LIN {X 0,Y 573.961,Z 401.905,A -85,B 0,C 180,E1 -2264.781,E2 -2264.781} C_VEL
LIN {X 0,Y 574.137,Z 387.873,A -85,B 0,C 180,E1 -2265.623,E2 -2265.623} C_VEL
LIN {X 0,Y 574.369,Z 373.799,A -85,B 0,C 180,E1 -2266.3,E2 -2266.3} C_VEL
LIN {X 0,Y 574.566,Z 359.304,A -85,B 0,C 180,E1 -2266.843,E2 -2266.843} C_VEL
LIN {X 0,Y 574.72,Z 343.895,A -85,B 0,C 180,E1 -2267.263,E2 -2267.263} C_VEL
LIN {X 0,Y 574.806,Z 328.514,A -85,B 0,C 180,E1 -2267.533,E2 -2267.533} C_VEL
LIN {X 0,Y 575.107,Z 176.129,A -85,B 0,C 180,E1 -2269.49,E2 -2269.49} C_VEL
LIN {X 0,Y 573.982,Z 170.376,A -85,B 0,C 180,E1 -2269.621,E2 -2269.621} C_VEL
LIN {X 0,Y 574.205,Z 150.282,A -85,B 0,C 180,E1 -2272.109,E2 -2272.109} C_VEL
LIN {X 0,Y 574.45,Z 130.828,A -85,B 0,C 180,E1 -2274.58,E2 -2274.58} C_VEL
LIN {X 0,Y 573.276,Z 124.83,A -85,B 0,C 180,E1 -2275.433,E2 -2275.433} C_VEL
LIN {X 0,Y 573.251,Z 124.698,A -85,B 0,C 180,E1 -2278.029,E2 -2278.029} C_VEL
LIN {X 0,Y 573.247,Z 124.707,A -85,B 0,C 180,E1 -2280.176,E2 -2280.176} C_VEL
LIN {X 0,Y 573.254,Z 124.699,A -85,B 0,C 180,E1 -2282.645,E2 -2282.645} C_VEL
LIN {X 0,Y 573.206,Z 124.704,A -85,B 0,C 180,E1 -2285.188,E2 -2285.188} C_VEL
LIN {X 0,Y 573.237,Z 124.707,A -85,B 0,C 180,E1 -2287.808,E2 -2287.808} C_VEL
LIN {X 0,Y 573.245,Z 124.7,A -85,B 0,C 180,E1 -2290.525,E2 -2290.525} C_VEL
LIN {X 0,Y 573.237,Z 124.702,A -85,B 0,C 180,E1 -2293.359,E2 -2293.359} C_VEL
LIN {X 0,Y 573.246,Z 124.701,A -85,B 0,C 180,E1 -2296.331,E2 -2296.331} C_VEL
LIN {X 0,Y 573.23,Z 124.698,A -85,B 0,C 180,E1 -2298.543,E2 -2298.543} C_VEL
LIN {X 0,Y 573.242,Z 124.702,A -85,B 0,C 180,E1 -2301.299,E2 -2301.299} C_VEL
LIN {X 0,Y 573.213,Z 124.704,A -85,B 0,C 180,E1 -2304.019,E2 -2304.019} C_VEL
LIN {X 0,Y 573.234,Z 124.694,A -85,B 0,C 180,E1 -2306.516,E2 -2306.516} C_VEL
LIN {X 0,Y 573.225,Z 124.703,A -85,B 0,C 180,E1 -2309.119,E2 -2309.119} C_VEL
LIN {X 0,Y 573.236,Z 124.707,A -85,B 0,C 180,E1 -2311.436,E2 -2311.436} C_VEL
LIN {X 0,Y 573.26,Z 124.697,A -85,B 0,C 180,E1 -2313.81,E2 -2313.81} C_VEL
LIN {X 0,Y 573.223,Z 124.702,A -85,B 0,C 180,E1 -2316.134,E2 -2316.134} C_VEL
LIN {X 0,Y 573.249,Z 124.706,A -85,B 0,C 180,E1 -2319.174,E2 -2319.174} C_VEL
LIN {X 0,Y 573.214,Z 124.707,A -85,B 0,C 180,E1 -2321.411,E2 -2321.411} C_VEL
LIN {X 0,Y 573.24,Z 124.699,A -85,B 0,C 180,E1 -2323.621,E2 -2323.621} C_VEL
LIN {X 0,Y 573.224,Z 124.705,A -85,B 0,C 180,E1 -2326.529,E2 -2326.529} C_VEL
LIN {X 0,Y 573.265,Z 124.705,A -85,B 0,C 180,E1 -2328.745,E2 -2328.745} C_VEL
LIN {X 0,Y 573.253,Z 124.697,A -85,B 0,C 180,E1 -2331.54,E2 -2331.54} C_VEL
LIN {X 0,Y 573.297,Z 124.697,A -85,B 0,C 180,E1 -2334.372,E2 -2334.372} C_VEL
LIN {X 0,Y 573.312,Z 124.69,A -85,B 0,C 180,E1 -2337.893,E2 -2337.893} C_VEL
LIN {X 0,Y 573.329,Z 124.693,A -85,B 0,C 180,E1 -2340.702,E2 -2340.702} C_VEL
LIN {X 0,Y 573.293,Z 124.695,A -85,B 0,C 180,E1 -2342.811,E2 -2342.811} C_VEL
LIN {X 0,Y 573.283,Z 124.695,A -85,B 0,C 180,E1 -2345.628,E2 -2345.628} C_VEL
LIN {X 0,Y 573.28,Z 124.699,A -85,B 0,C 180,E1 -2348.46,E2 -2348.46} C_VEL
LIN {X 0,Y 573.275,Z 124.695,A -85,B 0,C 180,E1 -2351.312,E2 -2351.312} C_VEL
LIN {X 0,Y 573.273,Z 124.698,A -85,B 0,C 180,E1 -2354.42,E2 -2354.42} C_VEL
LIN {X 0,Y 573.196,Z 124.705,A -85,B 0,C 180,E1 -2357.114,E2 -2357.114} C_VEL
LIN {X 0,Y 573.267,Z 124.696,A -85,B 0,C 180,E1 -2359.33,E2 -2359.33} C_VEL
LIN {X 0,Y 573.221,Z 124.705,A -85,B 0,C 180,E1 -2362.339,E2 -2362.339} C_VEL
LIN {X 0,Y 573.208,Z 124.704,A -85,B 0,C 180,E1 -2364.372,E2 -2364.372} C_VEL
LIN {X 0,Y 572.57,Z 124.783,A -85,B 0,C 180,E1 -2364.959,E2 -2364.959} C_VEL
LIN {X 0,Y 569.729,Z 125.144,A -85,B 0,C 180,E1 -2365.91,E2 -2365.91} C_VEL
LIN {X 0,Y 567.305,Z 125.446,A -85,B 0,C 180,E1 -2366.676,E2 -2366.676} C_VEL
LIN {X 0,Y 566.254,Z 125.574,A -85,B 0,C 180,E1 -2367.267,E2 -2367.267} C_VEL
LIN {X 0,Y 566.163,Z 125.584,A -85,B 0,C 180,E1 -2367.467,E2 -2367.467} C_VEL
LIN {X 0,Y 566.17,Z 125.584,A -85,B 0,C 180,E1 -2369.771,E2 -2369.771} C_VEL
LIN {X 0,Y 566.193,Z 125.57,A -85,B 0,C 180,E1 -2372.428,E2 -2372.428} C_VEL
LIN {X 0,Y 566.167,Z 125.581,A -85,B 0,C 180,E1 -2374.987,E2 -2374.987} C_VEL
LIN {X 0,Y 566.191,Z 125.585,A -85,B 0,C 180,E1 -2377.461,E2 -2377.461} C_VEL
LIN {X 0,Y 566.206,Z 125.57,A -85,B 0,C 180,E1 -2380.199,E2 -2380.199} C_VEL
LIN {X 0,Y 566.179,Z 125.584,A -85,B 0,C 180,E1 -2383.056,E2 -2383.056} C_VEL
LIN {X 0,Y 566.156,Z 125.579,A -85,B 0,C 180,E1 -2386.053,E2 -2386.053} C_VEL
LIN {X 0,Y 566.164,Z 125.587,A -85,B 0,C 180,E1 -2388.859,E2 -2388.859} C_VEL
LIN {X 0,Y 566.202,Z 125.581,A -85,B 0,C 180,E1 -2391.443,E2 -2391.443} C_VEL
LIN {X 0,Y 566.136,Z 125.585,A -85,B 0,C 180,E1 -2394.306,E2 -2394.306} C_VEL
LIN {X 0,Y 566.193,Z 125.585,A -85,B 0,C 180,E1 -2396.896,E2 -2396.896} C_VEL
LIN {X 0,Y 566.15,Z 125.578,A -85,B 0,C 180,E1 -2399.405,E2 -2399.405} C_VEL
LIN {X 0,Y 566.141,Z 125.586,A -85,B 0,C 180,E1 -2401.854,E2 -2401.854} C_VEL
LIN {X 0,Y 566.175,Z 125.585,A -85,B 0,C 180,E1 -2404.249,E2 -2404.249} C_VEL
LIN {X 0,Y 566.208,Z 125.751,A -85,B 0,C 180,E1 -2405.405,E2 -2405.405} C_VEL
LIN {X 0,Y 567.351,Z 131.059,A -85,B 0,C 180,E1 -2406.212,E2 -2406.212} C_VEL
LIN {X 0,Y 567.208,Z 146.629,A -85,B 0,C 180,E1 -2408.324,E2 -2408.324} C_VEL
LIN {X 0,Y 567.018,Z 160.677,A -85,B 0,C 180,E1 -2410.172,E2 -2410.172} C_VEL
LIN {X 0,Y 568.504,Z 168.273,A -85,B 0,C 180,E1 -2410.348,E2 -2410.348} C_VEL
LIN {X 0,Y 567.975,Z 326.141,A -85,B 0,C 180,E1 -2412.412,E2 -2412.412} C_VEL
LIN {X 0,Y 567.824,Z 341.766,A -85,B 0,C 180,E1 -2412.766,E2 -2412.766} C_VEL
LIN {X 0,Y 567.638,Z 357.075,A -85,B 0,C 180,E1 -2413.27,E2 -2413.27} C_VEL
LIN {X 0,Y 567.408,Z 371.73,A -85,B 0,C 180,E1 -2413.91,E2 -2413.91} C_VEL
LIN {X 0,Y 567.132,Z 385.048,A -85,B 0,C 180,E1 -2414.64,E2 -2414.64} C_VEL
LIN {X 0,Y 566.918,Z 397.981,A -85,B 0,C 180,E1 -2415.508,E2 -2415.508} C_VEL
LIN {X 0,Y 566.653,Z 410.889,A -85,B 0,C 180,E1 -2416.553,E2 -2416.553} C_VEL
LIN {X 0,Y 566.462,Z 422.085,A -85,B 0,C 180,E1 -2417.642,E2 -2417.642} C_VEL
LIN {X 0,Y 566.264,Z 432.178,A -85,B 0,C 180,E1 -2418.81,E2 -2418.81} C_VEL
LIN {X 0,Y 566.132,Z 442.003,A -85,B 0,C 180,E1 -2420.172,E2 -2420.172} C_VEL
LIN {X 0,Y 566.063,Z 449.494,A -85,B 0,C 180,E1 -2421.432,E2 -2421.432} C_VEL
LIN {X 0,Y 565.975,Z 456.499,A -85,B 0,C 180,E1 -2422.867,E2 -2422.867} C_VEL
LIN {X 0,Y 565.982,Z 462.009,A -85,B 0,C 180,E1 -2424.299,E2 -2424.299} C_VEL
LIN {X 0,Y 565.913,Z 466.177,A -85,B 0,C 180,E1 -2425.727,E2 -2425.727} C_VEL
LIN {X 0,Y 565.872,Z 469.112,A -85,B 0,C 180,E1 -2427.152,E2 -2427.152} C_VEL
LIN {X 0,Y 565.842,Z 470.879,A -85,B 0,C 180,E1 -2428.577,E2 -2428.577} C_VEL
LIN {X 0,Y 565.837,Z 471.496,A -85,B 0,C 180,E1 -2430,E2 -2430} C_VEL
LIN {X 0,Y 565.843,Z 470.941,A -85,B 0,C 180,E1 -2431.423,E2 -2431.423} C_VEL
LIN {X 0,Y 565.874,Z 469.257,A -85,B 0,C 180,E1 -2432.848,E2 -2432.848} C_VEL
LIN {X 0,Y 565.913,Z 466.404,A -85,B 0,C 180,E1 -2434.273,E2 -2434.273} C_VEL
LIN {X 0,Y 565.975,Z 462.318,A -85,B 0,C 180,E1 -2435.701,E2 -2435.701} C_VEL
LIN {X 0,Y 565.975,Z 456.903,A -85,B 0,C 180,E1 -2437.133,E2 -2437.133} C_VEL
LIN {X 0,Y 566.061,Z 450.002,A -85,B 0,C 180,E1 -2438.568,E2 -2438.568} C_VEL
LIN {X 0,Y 566.177,Z 441.393,A -85,B 0,C 180,E1 -2440.008,E2 -2440.008} C_VEL
LIN {X 0,Y 566.25,Z 432.953,A -85,B 0,C 180,E1 -2441.183,E2 -2441.183} C_VEL
LIN {X 0,Y 566.43,Z 422.913,A -85,B 0,C 180,E1 -2442.359,E2 -2442.359} C_VEL
LIN {X 0,Y 566.669,Z 410.869,A -85,B 0,C 180,E1 -2443.538,E2 -2443.538} C_VEL
LIN {X 0,Y 566.879,Z 399.242,A -85,B 0,C 180,E1 -2444.488,E2 -2444.488} C_VEL
LIN {X 0,Y 567.09,Z 386.467,A -85,B 0,C 180,E1 -2445.361,E2 -2445.361} C_VEL
LIN {X 0,Y 567.361,Z 373.456,A -85,B 0,C 180,E1 -2446.091,E2 -2446.091} C_VEL
LIN {X 0,Y 567.571,Z 359.261,A -85,B 0,C 180,E1 -2446.732,E2 -2446.732} C_VEL
LIN {X 0,Y 567.791,Z 344.711,A -85,B 0,C 180,E1 -2447.235,E2 -2447.235} C_VEL
LIN {X 0,Y 567.93,Z 329.3,A -85,B 0,C 180,E1 -2447.615,E2 -2447.615} C_VEL
LIN {X 0,Y 568.045,Z 307.857,A -85,B 0,C 180,E1 -2447.933,E2 -2447.933} C_VEL
LIN {X 0,Y 568.445,Z 167.858,A -85,B 0,C 180,E1 -2449.75,E2 -2449.75} C_VEL
LIN {X 0,Y 567.012,Z 160.622,A -85,B 0,C 180,E1 -2449.921,E2 -2449.921} C_VEL
LIN {X 0,Y 567.371,Z 139.147,A -85,B 0,C 180,E1 -2452.774,E2 -2452.774} C_VEL
LIN {X 0,Y 567.419,Z 131.697,A -85,B 0,C 180,E1 -2453.788,E2 -2453.788} C_VEL
LIN {X 0,Y 566.213,Z 125.822,A -85,B 0,C 180,E1 -2454.668,E2 -2454.668} C_VEL
LIN {X 0,Y 566.164,Z 125.581,A -85,B 0,C 180,E1 -2456.65,E2 -2456.65} C_VEL
LIN {X 0,Y 566.144,Z 125.58,A -85,B 0,C 180,E1 -2459.772,E2 -2459.772} C_VEL
LIN {X 0,Y 566.177,Z 125.581,A -85,B 0,C 180,E1 -2462.425,E2 -2462.425} C_VEL
LIN {X 0,Y 566.159,Z 125.589,A -85,B 0,C 180,E1 -2464.986,E2 -2464.986} C_VEL
LIN {X 0,Y 566.189,Z 125.582,A -85,B 0,C 180,E1 -2467.462,E2 -2467.462} C_VEL
LIN {X 0,Y 566.166,Z 125.579,A -85,B 0,C 180,E1 -2470.203,E2 -2470.203} C_VEL
LIN {X 0,Y 566.177,Z 125.584,A -85,B 0,C 180,E1 -2473.057,E2 -2473.057} C_VEL
LIN {X 0,Y 566.157,Z 125.582,A -85,B 0,C 180,E1 -2476.053,E2 -2476.053} C_VEL
LIN {X 0,Y 566.151,Z 125.584,A -85,B 0,C 180,E1 -2478.858,E2 -2478.858} C_VEL
LIN {X 0,Y 566.199,Z 125.575,A -85,B 0,C 180,E1 -2481.444,E2 -2481.444} C_VEL
LIN {X 0,Y 566.141,Z 125.59,A -85,B 0,C 180,E1 -2484.306,E2 -2484.306} C_VEL
LIN {X 0,Y 566.196,Z 125.573,A -85,B 0,C 180,E1 -2486.896,E2 -2486.896} C_VEL
LIN {X 0,Y 566.168,Z 125.576,A -85,B 0,C 180,E1 -2489.406,E2 -2489.406} C_VEL
LIN {X 0,Y 566.15,Z 125.585,A -85,B 0,C 180,E1 -2491.854,E2 -2491.854} C_VEL
LIN {X 0,Y 566.193,Z 125.585,A -85,B 0,C 180,E1 -2494.25,E2 -2494.25} C_VEL
LIN {X 0,Y 566.164,Z 125.581,A -85,B 0,C 180,E1 -2497.368,E2 -2497.368} C_VEL
LIN {X 0,Y 566.194,Z 125.579,A -85,B 0,C 180,E1 -2499.662,E2 -2499.662} C_VEL
LIN {X 0,Y 566.17,Z 125.586,A -85,B 0,C 180,E1 -2501.921,E2 -2501.921} C_VEL
LIN {X 0,Y 566.188,Z 125.576,A -85,B 0,C 180,E1 -2504.89,E2 -2504.89} C_VEL
LIN {X 0,Y 566.213,Z 125.582,A -85,B 0,C 180,E1 -2507.818,E2 -2507.818} C_VEL
LIN {X 0,Y 566.172,Z 125.585,A -85,B 0,C 180,E1 -2509.992,E2 -2509.992} C_VEL
LIN {X 0,Y 566.213,Z 125.574,A -85,B 0,C 180,E1 -2512.87,E2 -2512.87} C_VEL
LIN {X 0,Y 566.267,Z 125.569,A -85,B 0,C 180,E1 -2515.016,E2 -2515.016} C_VEL
LIN {X 0,Y 566.284,Z 125.569,A -85,B 0,C 180,E1 -2517.866,E2 -2517.866} C_VEL
LIN {X 0,Y 566.289,Z 125.565,A -85,B 0,C 180,E1 -2520.711,E2 -2520.711} C_VEL
LIN {X 0,Y 566.258,Z 125.569,A -85,B 0,C 180,E1 -2522.846,E2 -2522.846} C_VEL
LIN {X 0,Y 566.262,Z 125.573,A -85,B 0,C 180,E1 -2525.698,E2 -2525.698} C_VEL
LIN {X 0,Y 566.204,Z 125.575,A -85,B 0,C 180,E1 -2528.566,E2 -2528.566} C_VEL
LIN {X 0,Y 566.245,Z 125.577,A -85,B 0,C 180,E1 -2531.454,E2 -2531.454} C_VEL
LIN {X 0,Y 566.221,Z 125.574,A -85,B 0,C 180,E1 -2534.5,E2 -2534.5} C_VEL
LIN {X 0,Y 566.19,Z 125.583,A -85,B 0,C 180,E1 -2537.332,E2 -2537.332} C_VEL
LIN {X 0,Y 566.203,Z 125.577,A -85,B 0,C 180,E1 -2539.581,E2 -2539.581} C_VEL
LIN {X 0,Y 566.189,Z 125.577,A -85,B 0,C 180,E1 -2541.863,E2 -2541.863} C_VEL
LIN {X 0,Y 566.185,Z 125.583,A -85,B 0,C 180,E1 -2545.022,E2 -2545.022} C_VEL
LIN {X 0,Y 566.209,Z 125.577,A -85,B 0,C 180,E1 -2547.339,E2 -2547.339} C_VEL
LIN {X 0,Y 566.198,Z 125.576,A -85,B 0,C 180,E1 -2549.769,E2 -2549.769} C_VEL
LIN {X 0,Y 566.204,Z 125.578,A -85,B 0,C 180,E1 -2552.429,E2 -2552.429} C_VEL
LIN {X 0,Y 566.181,Z 125.581,A -85,B 0,C 180,E1 -2554.989,E2 -2554.989} C_VEL
LIN {X 0,Y 566.197,Z 125.577,A -85,B 0,C 180,E1 -2557.461,E2 -2557.461} C_VEL
LIN {X 0,Y 566.208,Z 125.579,A -85,B 0,C 180,E1 -2560.199,E2 -2560.199} C_VEL
LIN {X 0,Y 566.203,Z 125.577,A -85,B 0,C 180,E1 -2563.054,E2 -2563.054} C_VEL
LIN {X 0,Y 566.195,Z 125.582,A -85,B 0,C 180,E1 -2566.049,E2 -2566.049} C_VEL
LIN {X 0,Y 566.205,Z 125.576,A -85,B 0,C 180,E1 -2569.214,E2 -2569.214} C_VEL
LIN {X 0,Y 566.19,Z 125.58,A -85,B 0,C 180,E1 -2571.637,E2 -2571.637} C_VEL
LIN {X 0,Y 566.163,Z 125.586,A -85,B 0,C 180,E1 -2574.308,E2 -2574.308} C_VEL
LIN {X 0,Y 566.221,Z 125.572,A -85,B 0,C 180,E1 -2576.898,E2 -2576.898} C_VEL
LIN {X 0,Y 566.181,Z 125.58,A -85,B 0,C 180,E1 -2579.407,E2 -2579.407} C_VEL
LIN {X 0,Y 566.213,Z 125.574,A -85,B 0,C 180,E1 -2581.857,E2 -2581.857} C_VEL
LIN {X 0,Y 566.233,Z 125.711,A -85,B 0,C 180,E1 -2584.357,E2 -2584.357} C_VEL
LIN {X 0,Y 567.584,Z 132.266,A -85,B 0,C 180,E1 -2585.298,E2 -2585.298} C_VEL
LIN {X 0,Y 567.325,Z 151.718,A -85,B 0,C 180,E1 -2587.8,E2 -2587.8} C_VEL
LIN {X 0,Y 567.06,Z 170.307,A -85,B 0,C 180,E1 -2590.126,E2 -2590.126} C_VEL
LIN {X 0,Y 568.525,Z 178.114,A -85,B 0,C 180,E1 -2590.301,E2 -2590.301} C_VEL
LIN {X 0,Y 567.999,Z 335.64,A -85,B 0,C 180,E1 -2592.359,E2 -2592.359} C_VEL
LIN {X 0,Y 567.86,Z 351.148,A -85,B 0,C 180,E1 -2592.705,E2 -2592.705} C_VEL
LIN {X 0,Y 567.634,Z 365.796,A -85,B 0,C 180,E1 -2593.177,E2 -2593.177} C_VEL
LIN {X 0,Y 567.403,Z 380.776,A -85,B 0,C 180,E1 -2593.818,E2 -2593.818} C_VEL
LIN {X 0,Y 567.147,Z 394.249,A -85,B 0,C 180,E1 -2594.548,E2 -2594.548} C_VEL
LIN {X 0,Y 566.932,Z 406.519,A -85,B 0,C 180,E1 -2595.359,E2 -2595.359} C_VEL
LIN {X 0,Y 566.672,Z 419.292,A -85,B 0,C 180,E1 -2596.37,E2 -2596.37} C_VEL
LIN {X 0,Y 566.491,Z 430.749,A -85,B 0,C 180,E1 -2597.461,E2 -2597.461} C_VEL
LIN {X 0,Y 566.268,Z 441.311,A -85,B 0,C 180,E1 -2598.659,E2 -2598.659} C_VEL
LIN {X 0,Y 566.208,Z 449.855,A -85,B 0,C 180,E1 -2599.812,E2 -2599.812} C_VEL
LIN {X 0,Y 566.057,Z 457.735,A -85,B 0,C 180,E1 -2601.072,E2 -2601.072} C_VEL
LIN {X 0,Y 565.997,Z 465.09,A -85,B 0,C 180,E1 -2602.508,E2 -2602.508} C_VEL
LIN {X 0,Y 565.959,Z 470.922,A -85,B 0,C 180,E1 -2603.941,E2 -2603.941} C_VEL
LIN {X 0,Y 565.867,Z 474.386,A -85,B 0,C 180,E1 -2605.012,E2 -2605.012} C_VEL
LIN {X 0,Y 565.91,Z 477.889,A -85,B 0,C 180,E1 -2606.44,E2 -2606.44} C_VEL
LIN {X 0,Y 565.839,Z 480.191,A -85,B 0,C 180,E1 -2607.865,E2 -2607.865} C_VEL
LIN {X 0,Y 565.836,Z 481.349,A -85,B 0,C 180,E1 -2609.288,E2 -2609.288} C_VEL
LIN {X 0,Y 565.836,Z 481.348,A -85,B 0,C 180,E1 -2610.712,E2 -2610.712} C_VEL
LIN {X 0,Y 565.839,Z 480.189,A -85,B 0,C 180,E1 -2612.135,E2 -2612.135} C_VEL
LIN {X 0,Y 565.91,Z 477.886,A -85,B 0,C 180,E1 -2613.56,E2 -2613.56} C_VEL
LIN {X 0,Y 565.867,Z 474.386,A -85,B 0,C 180,E1 -2614.988,E2 -2614.988} C_VEL
LIN {X 0,Y 565.942,Z 469.609,A -85,B 0,C 180,E1 -2616.417,E2 -2616.417} C_VEL
LIN {X 0,Y 566.014,Z 463.422,A -85,B 0,C 180,E1 -2617.85,E2 -2617.85} C_VEL
LIN {X 0,Y 566.071,Z 455.646,A -85,B 0,C 180,E1 -2619.288,E2 -2619.288} C_VEL
LIN {X 0,Y 566.239,Z 447.368,A -85,B 0,C 180,E1 -2620.549,E2 -2620.549} C_VEL
LIN {X 0,Y 566.367,Z 437.391,A -85,B 0,C 180,E1 -2621.815,E2 -2621.815} C_VEL
LIN {X 0,Y 566.586,Z 427.186,A -85,B 0,C 180,E1 -2622.901,E2 -2622.901} C_VEL
LIN {X 0,Y 566.799,Z 415.019,A -85,B 0,C 180,E1 -2623.992,E2 -2623.992} C_VEL
LIN {X 0,Y 567.039,Z 402.337,A -85,B 0,C 180,E1 -2624.936,E2 -2624.936} C_VEL
LIN {X 0,Y 567.227,Z 389.508,A -85,B 0,C 180,E1 -2625.726,E2 -2625.726} C_VEL
LIN {X 0,Y 567.494,Z 374.824,A -85,B 0,C 180,E1 -2626.457,E2 -2626.457} C_VEL
LIN {X 0,Y 567.755,Z 360.613,A -85,B 0,C 180,E1 -2627.004,E2 -2627.004} C_VEL
LIN {X 0,Y 567.874,Z 346.147,A -85,B 0,C 180,E1 -2627.421,E2 -2627.421} C_VEL
LIN {X 0,Y 568.02,Z 330.546,A -85,B 0,C 180,E1 -2627.719,E2 -2627.719} C_VEL
LIN {X 0,Y 568.449,Z 177.138,A -85,B 0,C 180,E1 -2629.714,E2 -2629.714} C_VEL
LIN {X 0,Y 567.081,Z 170.463,A -85,B 0,C 180,E1 -2629.865,E2 -2629.865} C_VEL
LIN {X 0,Y 567.148,Z 159.516,A -85,B 0,C 180,E1 -2631.211,E2 -2631.211} C_VEL
LIN {X 0,Y 567.573,Z 138.034,A -85,B 0,C 180,E1 -2633.952,E2 -2633.952} C_VEL
LIN {X 0,Y 567.614,Z 132.265,A -85,B 0,C 180,E1 -2634.701,E2 -2634.701} C_VEL
LIN {X 0,Y 566.227,Z 125.676,A -85,B 0,C 180,E1 -2635.664,E2 -2635.664} C_VEL
LIN {X 0,Y 566.203,Z 125.576,A -85,B 0,C 180,E1 -2638.202,E2 -2638.202} C_VEL
LIN {X 0,Y 566.191,Z 125.575,A -85,B 0,C 180,E1 -2641.076,E2 -2641.076} C_VEL
LIN {X 0,Y 566.212,Z 125.578,A -85,B 0,C 180,E1 -2643.734,E2 -2643.734} C_VEL
LIN {X 0,Y 566.2,Z 125.579,A -85,B 0,C 180,E1 -2646.57,E2 -2646.57} C_VEL
LIN {X 0,Y 566.223,Z 125.578,A -85,B 0,C 180,E1 -2649.687,E2 -2649.687} C_VEL
LIN {X 0,Y 566.202,Z 125.575,A -85,B 0,C 180,E1 -2652.917,E2 -2652.917} C_VEL
LIN {X 0,Y 566.199,Z 125.582,A -85,B 0,C 180,E1 -2656.049,E2 -2656.049} C_VEL
LIN {X 0,Y 566.204,Z 125.576,A -85,B 0,C 180,E1 -2659.215,E2 -2659.215} C_VEL
LIN {X 0,Y 566.187,Z 125.587,A -85,B 0,C 180,E1 -2661.637,E2 -2661.637} C_VEL
LIN {X 0,Y 566.163,Z 125.58,A -85,B 0,C 180,E1 -2664.308,E2 -2664.308} C_VEL
LIN {X 0,Y 566.202,Z 125.571,A -85,B 0,C 180,E1 -2666.897,E2 -2666.897} C_VEL
LIN {X 0,Y 566.176,Z 125.586,A -85,B 0,C 180,E1 -2669.407,E2 -2669.407} C_VEL
LIN {X 0,Y 566.196,Z 125.579,A -85,B 0,C 180,E1 -2671.857,E2 -2671.857} C_VEL
LIN {X 0,Y 566.21,Z 125.573,A -85,B 0,C 180,E1 -2674.251,E2 -2674.251} C_VEL
LIN {X 0,Y 566.169,Z 125.584,A -85,B 0,C 180,E1 -2676.72,E2 -2676.72} C_VEL
LIN {X 0,Y 566.206,Z 125.576,A -85,B 0,C 180,E1 -2679.663,E2 -2679.663} C_VEL
LIN {X 0,Y 566.19,Z 125.582,A -85,B 0,C 180,E1 -2682.668,E2 -2682.668} C_VEL
LIN {X 0,Y 566.217,Z 125.574,A -85,B 0,C 180,E1 -2685.626,E2 -2685.626} C_VEL
LIN {X 0,Y 566.237,Z 125.579,A -85,B 0,C 180,E1 -2688.676,E2 -2688.676} C_VEL
LIN {X 0,Y 566.205,Z 125.576,A -85,B 0,C 180,E1 -2691.434,E2 -2691.434} C_VEL
LIN {X 0,Y 566.264,Z 125.572,A -85,B 0,C 180,E1 -2694.302,E2 -2694.302} C_VEL
LIN {X 0,Y 566.283,Z 125.565,A -85,B 0,C 180,E1 -2697.866,E2 -2697.866} C_VEL
LIN {X 0,Y 566.299,Z 125.568,A -85,B 0,C 180,E1 -2700.711,E2 -2700.711} C_VEL
LIN {X 0,Y 566.259,Z 125.571,A -85,B 0,C 180,E1 -2702.846,E2 -2702.846} C_VEL
LIN {X 0,Y 566.253,Z 125.571,A -85,B 0,C 180,E1 -2705.698,E2 -2705.698} C_VEL
LIN {X 0,Y 566.223,Z 125.576,A -85,B 0,C 180,E1 -2708.566,E2 -2708.566} C_VEL
LIN {X 0,Y 566.244,Z 125.572,A -85,B 0,C 180,E1 -2711.454,E2 -2711.454} C_VEL
LIN {X 0,Y 566.227,Z 125.574,A -85,B 0,C 180,E1 -2714.503,E2 -2714.503} C_VEL
LIN {X 0,Y 566.162,Z 125.582,A -85,B 0,C 180,E1 -2717.333,E2 -2717.333} C_VEL
LIN {X 0,Y 566.201,Z 125.579,A -85,B 0,C 180,E1 -2719.581,E2 -2719.581} C_VEL
LIN {X 0,Y 566.187,Z 125.586,A -85,B 0,C 180,E1 -2721.863,E2 -2721.863} C_VEL
LIN {X 0,Y 566.18,Z 125.578,A -85,B 0,C 180,E1 -2725.021,E2 -2725.021} C_VEL
LIN {X 0,Y 566.163,Z 125.584,A -85,B 0,C 180,E1 -2727.467,E2 -2727.467} C_VEL
LIN {X 0,Y 565.484,Z 125.67,A -85,B 0,C 180,E1 -2728.061,E2 -2728.061} C_VEL
LIN {X 0,Y 562.626,Z 126.023,A -85,B 0,C 180,E1 -2729.025,E2 -2729.025} C_VEL
LIN {X 0,Y 560.226,Z 126.324,A -85,B 0,C 180,E1 -2729.801,E2 -2729.801} C_VEL
LIN {X 0,Y 559.206,Z 126.444,A -85,B 0,C 180,E1 -2730.4,E2 -2730.4} C_VEL
LIN {X 0,Y 559.128,Z 126.453,A -85,B 0,C 180,E1 -2730.602,E2 -2730.602} C_VEL
LIN {X 0,Y 559.148,Z 126.446,A -85,B 0,C 180,E1 -2732.716,E2 -2732.716} C_VEL
LIN {X 0,Y 559.117,Z 126.464,A -85,B 0,C 180,E1 -2735.325,E2 -2735.325} C_VEL
LIN {X 0,Y 559.127,Z 126.457,A -85,B 0,C 180,E1 -2738.018,E2 -2738.018} C_VEL
LIN {X 0,Y 559.153,Z 126.449,A -85,B 0,C 180,E1 -2740.813,E2 -2740.813} C_VEL
LIN {X 0,Y 559.108,Z 126.463,A -85,B 0,C 180,E1 -2743.737,E2 -2743.737} C_VEL
LIN {X 0,Y 559.107,Z 126.457,A -85,B 0,C 180,E1 -2746.263,E2 -2746.263} C_VEL
LIN {X 0,Y 559.153,Z 126.46,A -85,B 0,C 180,E1 -2749.187,E2 -2749.187} C_VEL
LIN {X 0,Y 559.126,Z 126.459,A -85,B 0,C 180,E1 -2751.982,E2 -2751.982} C_VEL
LIN {X 0,Y 559.119,Z 126.465,A -85,B 0,C 180,E1 -2754.789,E2 -2754.789} C_VEL
LIN {X 0,Y 559.148,Z 126.459,A -85,B 0,C 180,E1 -2757.366,E2 -2757.366} C_VEL
LIN {X 0,Y 559.097,Z 126.456,A -85,B 0,C 180,E1 -2760.152,E2 -2760.152} C_VEL
LIN {X 0,Y 559.114,Z 126.458,A -85,B 0,C 180,E1 -2763.184,E2 -2763.184} C_VEL
LIN {X 0,Y 559.169,Z 126.704,A -85,B 0,C 180,E1 -2765.207,E2 -2765.207} C_VEL
LIN {X 0,Y 560.562,Z 133.52,A -85,B 0,C 180,E1 -2766.239,E2 -2766.239} C_VEL
LIN {X 0,Y 560.235,Z 152.686,A -85,B 0,C 180,E1 -2768.859,E2 -2768.859} C_VEL
LIN {X 0,Y 560.134,Z 160.746,A -85,B 0,C 180,E1 -2769.918,E2 -2769.918} C_VEL
LIN {X 0,Y 561.841,Z 169.153,A -85,B 0,C 180,E1 -2770.115,E2 -2770.115} C_VEL
LIN {X 0,Y 561.22,Z 326.422,A -85,B 0,C 180,E1 -2772.198,E2 -2772.198} C_VEL
LIN {X 0,Y 561.059,Z 341.789,A -85,B 0,C 180,E1 -2772.551,E2 -2772.551} C_VEL
LIN {X 0,Y 560.815,Z 357.088,A -85,B 0,C 180,E1 -2773.06,E2 -2773.06} C_VEL
LIN {X 0,Y 560.567,Z 371.737,A -85,B 0,C 180,E1 -2773.709,E2 -2773.709} C_VEL
LIN {X 0,Y 560.237,Z 385.059,A -85,B 0,C 180,E1 -2774.446,E2 -2774.446} C_VEL
LIN {X 0,Y 559.984,Z 398.392,A -85,B 0,C 180,E1 -2775.353,E2 -2775.353} C_VEL
LIN {X 0,Y 559.69,Z 410.896,A -85,B 0,C 180,E1 -2776.382,E2 -2776.382} C_VEL
LIN {X 0,Y 559.487,Z 422.09,A -85,B 0,C 180,E1 -2777.486,E2 -2777.486} C_VEL
LIN {X 0,Y 559.228,Z 432.788,A -85,B 0,C 180,E1 -2778.743,E2 -2778.743} C_VEL
LIN {X 0,Y 559.095,Z 442.006,A -85,B 0,C 180,E1 -2780.047,E2 -2780.047} C_VEL
LIN {X 0,Y 559.002,Z 449.496,A -85,B 0,C 180,E1 -2781.323,E2 -2781.323} C_VEL
LIN {X 0,Y 558.901,Z 456.501,A -85,B 0,C 180,E1 -2782.776,E2 -2782.776} C_VEL
LIN {X 0,Y 558.888,Z 462.011,A -85,B 0,C 180,E1 -2784.226,E2 -2784.226} C_VEL
LIN {X 0,Y 558.808,Z 466.178,A -85,B 0,C 180,E1 -2785.672,E2 -2785.672} C_VEL
LIN {X 0,Y 558.793,Z 469.112,A -85,B 0,C 180,E1 -2787.116,E2 -2787.116} C_VEL
LIN {X 0,Y 558.742,Z 470.878,A -85,B 0,C 180,E1 -2788.559,E2 -2788.559} C_VEL
LIN {X 0,Y 558.738,Z 471.496,A -85,B 0,C 180,E1 -2790,E2 -2790} C_VEL
LIN {X 0,Y 558.743,Z 470.94,A -85,B 0,C 180,E1 -2791.442,E2 -2791.442} C_VEL
LIN {X 0,Y 558.795,Z 469.255,A -85,B 0,C 180,E1 -2792.884,E2 -2792.884} C_VEL
LIN {X 0,Y 558.808,Z 466.403,A -85,B 0,C 180,E1 -2794.328,E2 -2794.328} C_VEL
LIN {X 0,Y 558.881,Z 462.316,A -85,B 0,C 180,E1 -2795.774,E2 -2795.774} C_VEL
LIN {X 0,Y 558.901,Z 456.9,A -85,B 0,C 180,E1 -2797.224,E2 -2797.224} C_VEL
LIN {X 0,Y 559.001,Z 449.998,A -85,B 0,C 180,E1 -2798.677,E2 -2798.677} C_VEL
LIN {X 0,Y 559.092,Z 442.572,A -85,B 0,C 180,E1 -2799.953,E2 -2799.953} C_VEL
LIN {X 0,Y 559.215,Z 433.511,A -85,B 0,C 180,E1 -2801.25,E2 -2801.25} C_VEL
LIN {X 0,Y 559.44,Z 422.908,A -85,B 0,C 180,E1 -2802.516,E2 -2802.516} C_VEL
LIN {X 0,Y 559.697,Z 410.863,A -85,B 0,C 180,E1 -2803.71,E2 -2803.71} C_VEL
LIN {X 0,Y 559.999,Z 398.172,A -85,B 0,C 180,E1 -2804.752,E2 -2804.752} C_VEL
LIN {X 0,Y 560.284,Z 385.006,A -85,B 0,C 180,E1 -2805.646,E2 -2805.646} C_VEL
LIN {X 0,Y 560.558,Z 371.676,A -85,B 0,C 180,E1 -2806.385,E2 -2806.385} C_VEL
LIN {X 0,Y 560.827,Z 356.983,A -85,B 0,C 180,E1 -2807.033,E2 -2807.033} C_VEL
LIN {X 0,Y 561.109,Z 341.475,A -85,B 0,C 180,E1 -2807.545,E2 -2807.545} C_VEL
LIN {X 0,Y 561.234,Z 326.429,A -85,B 0,C 180,E1 -2807.891,E2 -2807.891} C_VEL
LIN {X 0,Y 561.791,Z 168.927,A -85,B 0,C 180,E1 -2809.98,E2 -2809.98} C_VEL
LIN {X 0,Y 560.123,Z 160.807,A -85,B 0,C 180,E1 -2810.168,E2 -2810.168} C_VEL
LIN {X 0,Y 560.502,Z 140.614,A -85,B 0,C 180,E1 -2812.874,E2 -2812.874} C_VEL
LIN {X 0,Y 560.594,Z 134.103,A -85,B 0,C 180,E1 -2813.769,E2 -2813.769} C_VEL
LIN {X 0,Y 559.199,Z 126.935,A -85,B 0,C 180,E1 -2814.839,E2 -2814.839} C_VEL
LIN {X 0,Y 559.118,Z 126.491,A -85,B 0,C 180,E1 -2814.992,E2 -2814.992} C_VEL
LIN {X 0,Y 559.098,Z 126.468,A -85,B 0,C 180,E1 -2817.717,E2 -2817.717} C_VEL
LIN {X 0,Y 559.091,Z 126.455,A -85,B 0,C 180,E1 -2820.187,E2 -2820.187} C_VEL
LIN {X 0,Y 559.135,Z 126.461,A -85,B 0,C 180,E1 -2822.717,E2 -2822.717} C_VEL
LIN {X 0,Y 559.112,Z 126.465,A -85,B 0,C 180,E1 -2825.325,E2 -2825.325} C_VEL
LIN {X 0,Y 559.123,Z 126.459,A -85,B 0,C 180,E1 -2828.019,E2 -2828.019} C_VEL
LIN {X 0,Y 559.103,Z 126.465,A -85,B 0,C 180,E1 -2830.817,E2 -2830.817} C_VEL
LIN {X 0,Y 559.106,Z 126.457,A -85,B 0,C 180,E1 -2833.737,E2 -2833.737} C_VEL
LIN {X 0,Y 559.107,Z 126.462,A -85,B 0,C 180,E1 -2836.263,E2 -2836.263} C_VEL
LIN {X 0,Y 559.115,Z 126.455,A -85,B 0,C 180,E1 -2839.184,E2 -2839.184} C_VEL
LIN {X 0,Y 559.168,Z 126.452,A -85,B 0,C 180,E1 -2841.193,E2 -2841.193} C_VEL
LIN {X 0,Y 559.117,Z 126.46,A -85,B 0,C 180,E1 -2843.787,E2 -2843.787} C_VEL
LIN {X 0,Y 559.146,Z 126.458,A -85,B 0,C 180,E1 -2846.424,E2 -2846.424} C_VEL
LIN {X 0,Y 559.149,Z 126.452,A -85,B 0,C 180,E1 -2848.98,E2 -2848.98} C_VEL
LIN {X 0,Y 559.111,Z 126.46,A -85,B 0,C 180,E1 -2851.63,E2 -2851.63} C_VEL
LIN {X 0,Y 559.158,Z 126.457,A -85,B 0,C 180,E1 -2853.902,E2 -2853.902} C_VEL
LIN {X 0,Y 559.113,Z 126.46,A -85,B 0,C 180,E1 -2857.066,E2 -2857.066} C_VEL
LIN {X 0,Y 559.164,Z 126.452,A -85,B 0,C 180,E1 -2859.395,E2 -2859.395} C_VEL
LIN {X 0,Y 559.121,Z 126.461,A -85,B 0,C 180,E1 -2861.685,E2 -2861.685} C_VEL
LIN {X 0,Y 559.135,Z 126.455,A -85,B 0,C 180,E1 -2864.695,E2 -2864.695} C_VEL
LIN {X 0,Y 559.171,Z 126.457,A -85,B 0,C 180,E1 -2867.663,E2 -2867.663} C_VEL
LIN {X 0,Y 559.133,Z 126.464,A -85,B 0,C 180,E1 -2869.865,E2 -2869.865} C_VEL
LIN {X 0,Y 559.168,Z 126.451,A -85,B 0,C 180,E1 -2872.78,E2 -2872.78} C_VEL
LIN {X 0,Y 559.243,Z 126.444,A -85,B 0,C 180,E1 -2874.953,E2 -2874.953} C_VEL
LIN {X 0,Y 559.255,Z 126.445,A -85,B 0,C 180,E1 -2877.839,E2 -2877.839} C_VEL
LIN {X 0,Y 559.261,Z 126.441,A -85,B 0,C 180,E1 -2880.72,E2 -2880.72} C_VEL
LIN {X 0,Y 559.227,Z 126.445,A -85,B 0,C 180,E1 -2882.881,E2 -2882.881} C_VEL
LIN {X 0,Y 559.23,Z 126.448,A -85,B 0,C 180,E1 -2885.77,E2 -2885.77} C_VEL
LIN {X 0,Y 559.169,Z 126.452,A -85,B 0,C 180,E1 -2888.675,E2 -2888.675} C_VEL
LIN {X 0,Y 559.208,Z 126.451,A -85,B 0,C 180,E1 -2891.6,E2 -2891.6} C_VEL
LIN {X 0,Y 559.183,Z 126.452,A -85,B 0,C 180,E1 -2894.587,E2 -2894.587} C_VEL
LIN {X 0,Y 559.135,Z 126.459,A -85,B 0,C 180,E1 -2897.558,E2 -2897.558} C_VEL
LIN {X 0,Y 559.166,Z 126.452,A -85,B 0,C 180,E1 -2899.838,E2 -2899.838} C_VEL
LIN {X 0,Y 559.138,Z 126.455,A -85,B 0,C 180,E1 -2902.153,E2 -2902.153} C_VEL
LIN {X 0,Y 559.144,Z 126.457,A -85,B 0,C 180,E1 -2905.179,E2 -2905.179} C_VEL
LIN {X 0,Y 559.149,Z 126.455,A -85,B 0,C 180,E1 -2907.714,E2 -2907.714} C_VEL
LIN {X 0,Y 559.15,Z 126.457,A -85,B 0,C 180,E1 -2910.183,E2 -2910.183} C_VEL
LIN {X 0,Y 559.153,Z 126.452,A -85,B 0,C 180,E1 -2912.715,E2 -2912.715} C_VEL
LIN {X 0,Y 559.128,Z 126.457,A -85,B 0,C 180,E1 -2915.324,E2 -2915.324} C_VEL
LIN {X 0,Y 559.134,Z 126.46,A -85,B 0,C 180,E1 -2918.017,E2 -2918.017} C_VEL
LIN {X 0,Y 559.156,Z 126.454,A -85,B 0,C 180,E1 -2920.812,E2 -2920.812} C_VEL
LIN {X 0,Y 559.142,Z 126.458,A -85,B 0,C 180,E1 -2923.734,E2 -2923.734} C_VEL
LIN {X 0,Y 559.146,Z 126.456,A -85,B 0,C 180,E1 -2926.804,E2 -2926.804} C_VEL
LIN {X 0,Y 559.156,Z 126.454,A -85,B 0,C 180,E1 -2929.187,E2 -2929.187} C_VEL
LIN {X 0,Y 559.136,Z 126.464,A -85,B 0,C 180,E1 -2931.982,E2 -2931.982} C_VEL
LIN {X 0,Y 559.132,Z 126.458,A -85,B 0,C 180,E1 -2934.787,E2 -2934.787} C_VEL
LIN {X 0,Y 559.157,Z 126.454,A -85,B 0,C 180,E1 -2937.364,E2 -2937.364} C_VEL
LIN {X 0,Y 559.15,Z 126.461,A -85,B 0,C 180,E1 -2940.142,E2 -2940.142} C_VEL
LIN {X 0,Y 559.17,Z 126.456,A -85,B 0,C 180,E1 -2943.098,E2 -2943.098} C_VEL
LIN {X 0,Y 559.218,Z 126.664,A -85,B 0,C 180,E1 -2944.155,E2 -2944.155} C_VEL
LIN {X 0,Y 560.72,Z 133.702,A -85,B 0,C 180,E1 -2945.173,E2 -2945.173} C_VEL
LIN {X 0,Y 560.451,Z 153.154,A -85,B 0,C 180,E1 -2947.708,E2 -2947.708} C_VEL
LIN {X 0,Y 560.152,Z 170.128,A -85,B 0,C 180,E1 -2949.864,E2 -2949.864} C_VEL
LIN {X 0,Y 561.843,Z 179.314,A -85,B 0,C 180,E1 -2950.074,E2 -2950.074} C_VEL
LIN {X 0,Y 561.257,Z 335.486,A -85,B 0,C 180,E1 -2952.138,E2 -2952.138} C_VEL
LIN {X 0,Y 561.095,Z 350.687,A -85,B 0,C 180,E1 -2952.478,E2 -2952.478} C_VEL
LIN {X 0,Y 560.83,Z 365.797,A -85,B 0,C 180,E1 -2952.967,E2 -2952.967} C_VEL
LIN {X 0,Y 560.563,Z 380.78,A -85,B 0,C 180,E1 -2953.615,E2 -2953.615} C_VEL
LIN {X 0,Y 560.283,Z 394.252,A -85,B 0,C 180,E1 -2954.354,E2 -2954.354} C_VEL
LIN {X 0,Y 559.998,Z 407.302,A -85,B 0,C 180,E1 -2955.23,E2 -2955.23} C_VEL
LIN {X 0,Y 559.697,Z 420.353,A -85,B 0,C 180,E1 -2956.29,E2 -2956.29} C_VEL
LIN {X 0,Y 559.474,Z 432.508,A -85,B 0,C 180,E1 -2957.485,E2 -2957.485} C_VEL
LIN {X 0,Y 559.197,Z 443.244,A -85,B 0,C 180,E1 -2958.758,E2 -2958.758} C_VEL
LIN {X 0,Y 559.092,Z 452.295,A -85,B 0,C 180,E1 -2960.047,E2 -2960.047} C_VEL
LIN {X 0,Y 559,Z 459.75,A -85,B 0,C 180,E1 -2961.323,E2 -2961.323} C_VEL
LIN {X 0,Y 558.899,Z 466.7,A -85,B 0,C 180,E1 -2962.776,E2 -2962.776} C_VEL
LIN {X 0,Y 558.888,Z 472.162,A -85,B 0,C 180,E1 -2964.226,E2 -2964.226} C_VEL
LIN {X 0,Y 558.809,Z 476.291,A -85,B 0,C 180,E1 -2965.672,E2 -2965.672} C_VEL
LIN {X 0,Y 558.793,Z 479.185,A -85,B 0,C 180,E1 -2967.116,E2 -2967.116} C_VEL
LIN {X 0,Y 558.742,Z 480.91,A -85,B 0,C 180,E1 -2968.558,E2 -2968.558} C_VEL
LIN {X 0,Y 558.737,Z 481.5,A -85,B 0,C 180,E1 -2970,E2 -2970} C_VEL
LIN {X 0,Y 558.742,Z 480.908,A -85,B 0,C 180,E1 -2971.441,E2 -2971.441} C_VEL
LIN {X 0,Y 558.793,Z 479.182,A -85,B 0,C 180,E1 -2972.884,E2 -2972.884} C_VEL
LIN {X 0,Y 558.808,Z 476.289,A -85,B 0,C 180,E1 -2974.328,E2 -2974.328} C_VEL
LIN {X 0,Y 558.888,Z 472.165,A -85,B 0,C 180,E1 -2975.774,E2 -2975.774} C_VEL
LIN {X 0,Y 558.899,Z 466.701,A -85,B 0,C 180,E1 -2977.224,E2 -2977.224} C_VEL
LIN {X 0,Y 559,Z 459.745,A -85,B 0,C 180,E1 -2978.677,E2 -2978.677} C_VEL
LIN {X 0,Y 559.091,Z 452.292,A -85,B 0,C 180,E1 -2979.953,E2 -2979.953} C_VEL
LIN {X 0,Y 559.227,Z 443.125,A -85,B 0,C 180,E1 -2981.257,E2 -2981.257} C_VEL
LIN {X 0,Y 559.474,Z 432.508,A -85,B 0,C 180,E1 -2982.515,E2 -2982.515} C_VEL
LIN {X 0,Y 559.701,Z 420.359,A -85,B 0,C 180,E1 -2983.71,E2 -2983.71} C_VEL
LIN {X 0,Y 560.005,Z 407.531,A -85,B 0,C 180,E1 -2984.754,E2 -2984.754} C_VEL
LIN {X 0,Y 560.284,Z 394.251,A -85,B 0,C 180,E1 -2985.646,E2 -2985.646} C_VEL
LIN {X 0,Y 560.562,Z 380.773,A -85,B 0,C 180,E1 -2986.385,E2 -2986.385} C_VEL
LIN {X 0,Y 560.855,Z 365.81,A -85,B 0,C 180,E1 -2987.032,E2 -2987.032} C_VEL
LIN {X 0,Y 561.062,Z 350.725,A -85,B 0,C 180,E1 -2987.522,E2 -2987.522} C_VEL
LIN {X 0,Y 561.238,Z 335.242,A -85,B 0,C 180,E1 -2987.866,E2 -2987.866} C_VEL
LIN {X 0,Y 561.774,Z 178.38,A -85,B 0,C 180,E1 -2989.941,E2 -2989.941} C_VEL
LIN {X 0,Y 560.16,Z 170.234,A -85,B 0,C 180,E1 -2990.13,E2 -2990.13} C_VEL
LIN {X 0,Y 560.441,Z 150.16,A -85,B 0,C 180,E1 -2992.682,E2 -2992.682} C_VEL
LIN {X 0,Y 560.731,Z 133.703,A -85,B 0,C 180,E1 -2994.827,E2 -2994.827} C_VEL
LIN {X 0,Y 559.201,Z 126.58,A -85,B 0,C 180,E1 -2995.871,E2 -2995.871} C_VEL
LIN {X 0,Y 559.164,Z 126.455,A -85,B 0,C 180,E1 -2998.53,E2 -2998.53} C_VEL
LIN {X 0,Y 559.146,Z 126.452,A -85,B 0,C 180,E1 -3001.273,E2 -3001.273} C_VEL
LIN {X 0,Y 559.166,Z 126.459,A -85,B 0,C 180,E1 -3003.949,E2 -3003.949} C_VEL
LIN {X 0,Y 559.141,Z 126.456,A -85,B 0,C 180,E1 -3007.108,E2 -3007.108} C_VEL
LIN {X 0,Y 559.166,Z 126.459,A -85,B 0,C 180,E1 -3009.942,E2 -3009.942} C_VEL
LIN {X 0,Y 559.158,Z 126.453,A -85,B 0,C 180,E1 -3012.744,E2 -3012.744} C_VEL
LIN {X 0,Y 559.153,Z 126.463,A -85,B 0,C 180,E1 -3015.761,E2 -3015.761} C_VEL
LIN {X 0,Y 559.164,Z 126.452,A -85,B 0,C 180,E1 -3018.23,E2 -3018.23} C_VEL
LIN {X 0,Y 559.175,Z 126.452,A -85,B 0,C 180,E1 -3021.192,E2 -3021.192} C_VEL
LIN {X 0,Y 559.14,Z 126.46,A -85,B 0,C 180,E1 -3023.789,E2 -3023.789} C_VEL
LIN {X 0,Y 559.147,Z 126.447,A -85,B 0,C 180,E1 -3026.424,E2 -3026.424} C_VEL
LIN {X 0,Y 559.153,Z 126.453,A -85,B 0,C 180,E1 -3028.981,E2 -3028.981} C_VEL
LIN {X 0,Y 559.17,Z 126.457,A -85,B 0,C 180,E1 -3031.619,E2 -3031.619} C_VEL
LIN {X 0,Y 559.179,Z 126.45,A -85,B 0,C 180,E1 -3033.903,E2 -3033.903} C_VEL
LIN {X 0,Y 559.138,Z 126.458,A -85,B 0,C 180,E1 -3036.572,E2 -3036.572} C_VEL
LIN {X 0,Y 559.176,Z 126.455,A -85,B 0,C 180,E1 -3039.395,E2 -3039.395} C_VEL
LIN {X 0,Y 559.132,Z 126.458,A -85,B 0,C 180,E1 -3041.685,E2 -3041.685} C_VEL
LIN {X 0,Y 559.156,Z 126.451,A -85,B 0,C 180,E1 -3043.948,E2 -3043.948} C_VEL
LIN {X 0,Y 559.16,Z 126.453,A -85,B 0,C 180,E1 -3046.184,E2 -3046.184} C_VEL
LIN {X 0,Y 559.208,Z 126.454,A -85,B 0,C 180,E1 -3048.605,E2 -3048.605} C_VEL
LIN {X 0,Y 559.17,Z 126.453,A -85,B 0,C 180,E1 -3051.325,E2 -3051.325} C_VEL
LIN {X 0,Y 559.232,Z 126.447,A -85,B 0,C 180,E1 -3054.23,E2 -3054.23} C_VEL
LIN {X 0,Y 559.254,Z 126.441,A -85,B 0,C 180,E1 -3057.84,E2 -3057.84} C_VEL
LIN {X 0,Y 559.27,Z 126.443,A -85,B 0,C 180,E1 -3060.72,E2 -3060.72} C_VEL
LIN {X 0,Y 559.225,Z 126.446,A -85,B 0,C 180,E1 -3062.882,E2 -3062.882} C_VEL
LIN {X 0,Y 559.223,Z 126.447,A -85,B 0,C 180,E1 -3065.77,E2 -3065.77} C_VEL
LIN {X 0,Y 559.182,Z 126.452,A -85,B 0,C 180,E1 -3068.675,E2 -3068.675} C_VEL
LIN {X 0,Y 559.206,Z 126.45,A -85,B 0,C 180,E1 -3071.6,E2 -3071.6} C_VEL
LIN {X 0,Y 559.183,Z 126.451,A -85,B 0,C 180,E1 -3074.588,E2 -3074.588} C_VEL
LIN {X 0,Y 559.117,Z 126.462,A -85,B 0,C 180,E1 -3077.558,E2 -3077.558} C_VEL
LIN {X 0,Y 559.164,Z 126.459,A -85,B 0,C 180,E1 -3079.838,E2 -3079.838} C_VEL
LIN {X 0,Y 559.133,Z 126.462,A -85,B 0,C 180,E1 -3082.153,E2 -3082.153} C_VEL
LIN {X 0,Y 559.14,Z 126.455,A -85,B 0,C 180,E1 -3085.178,E2 -3085.178} C_VEL
LIN {X 0,Y 559.12,Z 126.468,A -85,B 0,C 180,E1 -3087.716,E2 -3087.716} C_VEL
LIN {X 0,Y 559.128,Z 126.453,A -85,B 0,C 180,E1 -3090.602,E2 -3090.602} C_VEL
LIN {X 0,Y 558.471,Z 126.54,A -85,B 0,C 180,E1 -3091.204,E2 -3091.204} C_VEL
LIN {X 0,Y 555.611,Z 126.888,A -85,B 0,C 180,E1 -3092.18,E2 -3092.18} C_VEL
LIN {X 0,Y 553.193,Z 127.188,A -85,B 0,C 180,E1 -3092.966,E2 -3092.966} C_VEL
LIN {X 0,Y 552.164,Z 127.325,A -85,B 0,C 180,E1 -3093.572,E2 -3093.572} C_VEL
LIN {X 0,Y 552.086,Z 127.331,A -85,B 0,C 180,E1 -3093.778,E2 -3093.778} C_VEL
LIN {X 0,Y 552.098,Z 127.335,A -85,B 0,C 180,E1 -3096.748,E2 -3096.748} C_VEL
LIN {X 0,Y 552.126,Z 127.328,A -85,B 0,C 180,E1 -3099.528,E2 -3099.528} C_VEL
LIN {X 0,Y 552.086,Z 127.334,A -85,B 0,C 180,E1 -3102.43,E2 -3102.43} C_VEL
LIN {X 0,Y 552.075,Z 127.337,A -85,B 0,C 180,E1 -3105.56,E2 -3105.56} C_VEL
LIN {X 0,Y 552.076,Z 127.34,A -85,B 0,C 180,E1 -3108.684,E2 -3108.684} C_VEL
LIN {X 0,Y 552.112,Z 127.336,A -85,B 0,C 180,E1 -3111.411,E2 -3111.411} C_VEL
LIN {X 0,Y 552.068,Z 127.336,A -85,B 0,C 180,E1 -3114.155,E2 -3114.155} C_VEL
LIN {X 0,Y 552.106,Z 127.339,A -85,B 0,C 180,E1 -3117.155,E2 -3117.155} C_VEL
LIN {X 0,Y 552.068,Z 127.329,A -85,B 0,C 180,E1 -3119.959,E2 -3119.959} C_VEL
LIN {X 0,Y 552.077,Z 127.334,A -85,B 0,C 180,E1 -3123.013,E2 -3123.013} C_VEL
LIN {X 0,Y 552.12,Z 127.429,A -85,B 0,C 180,E1 -3124.936,E2 -3124.936} C_VEL
LIN {X 0,Y 553.329,Z 132.95,A -85,B 0,C 180,E1 -3125.819,E2 -3125.819} C_VEL
LIN {X 0,Y 553.702,Z 137.287,A -85,B 0,C 180,E1 -3126.446,E2 -3126.446} C_VEL
LIN {X 0,Y 553.239,Z 158.274,A -85,B 0,C 180,E1 -3129.339,E2 -3129.339} C_VEL
LIN {X 0,Y 553.279,Z 161.046,A -85,B 0,C 180,E1 -3129.672,E2 -3129.672} C_VEL
LIN {X 0,Y 555.178,Z 170.647,A -85,B 0,C 180,E1 -3129.885,E2 -3129.885} C_VEL
LIN {X 0,Y 554.468,Z 326.232,A -85,B 0,C 180,E1 -3131.968,E2 -3131.968} C_VEL
LIN {X 0,Y 554.292,Z 341.875,A -85,B 0,C 180,E1 -3132.331,E2 -3132.331} C_VEL
LIN {X 0,Y 554.031,Z 357.16,A -85,B 0,C 180,E1 -3132.847,E2 -3132.847} C_VEL
LIN {X 0,Y 553.741,Z 371.79,A -85,B 0,C 180,E1 -3133.502,E2 -3133.502} C_VEL
LIN {X 0,Y 553.374,Z 385.096,A -85,B 0,C 180,E1 -3134.248,E2 -3134.248} C_VEL
LIN {X 0,Y 553.063,Z 398.736,A -85,B 0,C 180,E1 -3135.191,E2 -3135.191} C_VEL
LIN {X 0,Y 552.723,Z 410.903,A -85,B 0,C 180,E1 -3136.207,E2 -3136.207} C_VEL
LIN {X 0,Y 552.489,Z 422.096,A -85,B 0,C 180,E1 -3137.324,E2 -3137.324} C_VEL
LIN {X 0,Y 552.199,Z 433.342,A -85,B 0,C 180,E1 -3138.672,E2 -3138.672} C_VEL
LIN {X 0,Y 552.075,Z 442.009,A -85,B 0,C 180,E1 -3139.919,E2 -3139.919} C_VEL
LIN {X 0,Y 551.92,Z 449.498,A -85,B 0,C 180,E1 -3141.211,E2 -3141.211} C_VEL
LIN {X 0,Y 551.821,Z 456.503,A -85,B 0,C 180,E1 -3142.683,E2 -3142.683} C_VEL
LIN {X 0,Y 551.796,Z 462.013,A -85,B 0,C 180,E1 -3144.152,E2 -3144.152} C_VEL
LIN {X 0,Y 551.706,Z 466.179,A -85,B 0,C 180,E1 -3145.617,E2 -3145.617} C_VEL
LIN {X 0,Y 551.717,Z 469.111,A -85,B 0,C 180,E1 -3147.079,E2 -3147.079} C_VEL
LIN {X 0,Y 551.641,Z 470.878,A -85,B 0,C 180,E1 -3148.54,E2 -3148.54} C_VEL
LIN {X 0,Y 551.638,Z 471.496,A -85,B 0,C 180,E1 -3150,E2 -3150} C_VEL
LIN {X 0,Y 551.643,Z 470.939,A -85,B 0,C 180,E1 -3151.46,E2 -3151.46} C_VEL
LIN {X 0,Y 551.719,Z 469.254,A -85,B 0,C 180,E1 -3152.921,E2 -3152.921} C_VEL
LIN {X 0,Y 551.705,Z 466.401,A -85,B 0,C 180,E1 -3154.384,E2 -3154.384} C_VEL
LIN {X 0,Y 551.787,Z 462.314,A -85,B 0,C 180,E1 -3155.848,E2 -3155.848} C_VEL
LIN {X 0,Y 551.821,Z 456.897,A -85,B 0,C 180,E1 -3157.317,E2 -3157.317} C_VEL
LIN {X 0,Y 551.919,Z 449.995,A -85,B 0,C 180,E1 -3158.79,E2 -3158.79} C_VEL
LIN {X 0,Y 552.071,Z 442.569,A -85,B 0,C 180,E1 -3160.081,E2 -3160.081} C_VEL
LIN {X 0,Y 552.184,Z 434.057,A -85,B 0,C 180,E1 -3161.32,E2 -3161.32} C_VEL
LIN {X 0,Y 552.395,Z 424.529,A -85,B 0,C 180,E1 -3162.491,E2 -3162.491} C_VEL
LIN {X 0,Y 552.673,Z 413.793,A -85,B 0,C 180,E1 -3163.607,E2 -3163.607} C_VEL
LIN {X 0,Y 552.97,Z 402.081,A -85,B 0,C 180,E1 -3164.632,E2 -3164.632} C_VEL
LIN {X 0,Y 553.278,Z 389.315,A -85,B 0,C 180,E1 -3165.566,E2 -3165.566} C_VEL
LIN {X 0,Y 553.651,Z 375.235,A -85,B 0,C 180,E1 -3166.406,E2 -3166.406} C_VEL
LIN {X 0,Y 553.943,Z 360.413,A -85,B 0,C 180,E1 -3167.109,E2 -3167.109} C_VEL
LIN {X 0,Y 554.249,Z 344.737,A -85,B 0,C 180,E1 -3167.67,E2 -3167.67} C_VEL
LIN {X 0,Y 554.41,Z 329.386,A -85,B 0,C 180,E1 -3168.058,E2 -3168.058} C_VEL
LIN {X 0,Y 554.562,Z 307.729,A -85,B 0,C 180,E1 -3168.386,E2 -3168.386} C_VEL
LIN {X 0,Y 555.143,Z 170.095,A -85,B 0,C 180,E1 -3170.214,E2 -3170.214} C_VEL
LIN {X 0,Y 553.24,Z 161.009,A -85,B 0,C 180,E1 -3170.421,E2 -3170.421} C_VEL
LIN {X 0,Y 553.345,Z 153.416,A -85,B 0,C 180,E1 -3171.417,E2 -3171.417} C_VEL
LIN {X 0,Y 553.759,Z 136.084,A -85,B 0,C 180,E1 -3173.809,E2 -3173.809} C_VEL
LIN {X 0,Y 552.843,Z 130.76,A -85,B 0,C 180,E1 -3174.603,E2 -3174.603} C_VEL
LIN {X 0,Y 552.119,Z 127.507,A -85,B 0,C 180,E1 -3175.136,E2 -3175.136} C_VEL
LIN {X 0,Y 552.047,Z 127.343,A -85,B 0,C 180,E1 -3178.102,E2 -3178.102} C_VEL
LIN {X 0,Y 552.067,Z 127.33,A -85,B 0,C 180,E1 -3180.612,E2 -3180.612} C_VEL
LIN {X 0,Y 552.095,Z 127.341,A -85,B 0,C 180,E1 -3183.187,E2 -3183.187} C_VEL
LIN {X 0,Y 552.067,Z 127.337,A -85,B 0,C 180,E1 -3185.845,E2 -3185.845} C_VEL
LIN {X 0,Y 552.11,Z 127.336,A -85,B 0,C 180,E1 -3188.59,E2 -3188.59} C_VEL
LIN {X 0,Y 552.063,Z 127.341,A -85,B 0,C 180,E1 -3191.451,E2 -3191.451} C_VEL
LIN {X 0,Y 552.075,Z 127.337,A -85,B 0,C 180,E1 -3194.529,E2 -3194.529} C_VEL
LIN {X 0,Y 552.083,Z 127.335,A -85,B 0,C 180,E1 -3197.59,E2 -3197.59} C_VEL
LIN {X 0,Y 552.122,Z 127.328,A -85,B 0,C 180,E1 -3200.472,E2 -3200.472} C_VEL
LIN {X 0,Y 552.099,Z 127.335,A -85,B 0,C 180,E1 -3203.318,E2 -3203.318} C_VEL
LIN {X 0,Y 552.098,Z 127.333,A -85,B 0,C 180,E1 -3205.937,E2 -3205.937} C_VEL
LIN {X 0,Y 552.105,Z 127.33,A -85,B 0,C 180,E1 -3208.54,E2 -3208.54} C_VEL
LIN {X 0,Y 552.08,Z 127.335,A -85,B 0,C 180,E1 -3211.447,E2 -3211.447} C_VEL
LIN {X 0,Y 552.084,Z 127.34,A -85,B 0,C 180,E1 -3214.353,E2 -3214.353} C_VEL
LIN {X 0,Y 552.09,Z 127.336,A -85,B 0,C 180,E1 -3216.757,E2 -3216.757} C_VEL
LIN {X 0,Y 552.107,Z 127.33,A -85,B 0,C 180,E1 -3219.119,E2 -3219.119} C_VEL
LIN {X 0,Y 552.082,Z 127.335,A -85,B 0,C 180,E1 -3221.443,E2 -3221.443} C_VEL
LIN {X 0,Y 552.092,Z 127.334,A -85,B 0,C 180,E1 -3224.495,E2 -3224.495} C_VEL
LIN {X 0,Y 552.11,Z 127.331,A -85,B 0,C 180,E1 -3226.754,E2 -3226.754} C_VEL
LIN {X 0,Y 552.163,Z 127.325,A -85,B 0,C 180,E1 -3228.993,E2 -3228.993} C_VEL
LIN {X 0,Y 552.147,Z 127.332,A -85,B 0,C 180,E1 -3231.951,E2 -3231.951} C_VEL
LIN {X 0,Y 552.219,Z 127.319,A -85,B 0,C 180,E1 -3234.889,E2 -3234.889} C_VEL
LIN {X 0,Y 552.226,Z 127.321,A -85,B 0,C 180,E1 -3237.812,E2 -3237.812} C_VEL
LIN {X 0,Y 552.233,Z 127.316,A -85,B 0,C 180,E1 -3240.729,E2 -3240.729} C_VEL
LIN {X 0,Y 552.195,Z 127.321,A -85,B 0,C 180,E1 -3242.918,E2 -3242.918} C_VEL
LIN {X 0,Y 552.199,Z 127.323,A -85,B 0,C 180,E1 -3245.844,E2 -3245.844} C_VEL
LIN {X 0,Y 552.141,Z 127.329,A -85,B 0,C 180,E1 -3248.786,E2 -3248.786} C_VEL
LIN {X 0,Y 552.164,Z 127.327,A -85,B 0,C 180,E1 -3251.75,E2 -3251.75} C_VEL
LIN {X 0,Y 552.131,Z 127.332,A -85,B 0,C 180,E1 -3254.748,E2 -3254.748} C_VEL
LIN {X 0,Y 552.094,Z 127.334,A -85,B 0,C 180,E1 -3257.789,E2 -3257.789} C_VEL
LIN {X 0,Y 552.127,Z 127.328,A -85,B 0,C 180,E1 -3260.101,E2 -3260.101} C_VEL
LIN {X 0,Y 552.089,Z 127.336,A -85,B 0,C 180,E1 -3262.451,E2 -3262.451} C_VEL
LIN {X 0,Y 552.113,Z 127.329,A -85,B 0,C 180,E1 -3265.645,E2 -3265.645} C_VEL
LIN {X 0,Y 552.126,Z 127.337,A -85,B 0,C 180,E1 -3268.562,E2 -3268.562} C_VEL
LIN {X 0,Y 552.113,Z 127.326,A -85,B 0,C 180,E1 -3271.475,E2 -3271.475} C_VEL
LIN {X 0,Y 552.126,Z 127.325,A -85,B 0,C 180,E1 -3274.169,E2 -3274.169} C_VEL
LIN {X 0,Y 552.106,Z 127.338,A -85,B 0,C 180,E1 -3276.747,E2 -3276.747} C_VEL
LIN {X 0,Y 552.131,Z 127.325,A -85,B 0,C 180,E1 -3279.527,E2 -3279.527} C_VEL
LIN {X 0,Y 552.131,Z 127.338,A -85,B 0,C 180,E1 -3282.425,E2 -3282.425} C_VEL
LIN {X 0,Y 552.095,Z 127.332,A -85,B 0,C 180,E1 -3285.562,E2 -3285.562} C_VEL
LIN {X 0,Y 552.122,Z 127.334,A -85,B 0,C 180,E1 -3288.554,E2 -3288.554} C_VEL
LIN {X 0,Y 552.121,Z 127.33,A -85,B 0,C 180,E1 -3291.411,E2 -3291.411} C_VEL
LIN {X 0,Y 552.086,Z 127.34,A -85,B 0,C 180,E1 -3294.156,E2 -3294.156} C_VEL
LIN {X 0,Y 552.116,Z 127.329,A -85,B 0,C 180,E1 -3296.814,E2 -3296.814} C_VEL
LIN {X 0,Y 552.103,Z 127.332,A -85,B 0,C 180,E1 -3299.391,E2 -3299.391} C_VEL
LIN {X 0,Y 552.11,Z 127.327,A -85,B 0,C 180,E1 -3301.902,E2 -3301.902} C_VEL
LIN {X 0,Y 552.194,Z 127.541,A -85,B 0,C 180,E1 -3303.928,E2 -3303.928} C_VEL
LIN {X 0,Y 553.869,Z 135.226,A -85,B 0,C 180,E1 -3305.057,E2 -3305.057} C_VEL
LIN {X 0,Y 553.569,Z 154.591,A -85,B 0,C 180,E1 -3307.612,E2 -3307.612} C_VEL
LIN {X 0,Y 553.304,Z 170.308,A -85,B 0,C 180,E1 -3309.62,E2 -3309.62} C_VEL
LIN {X 0,Y 555.168,Z 180.291,A -85,B 0,C 180,E1 -3309.838,E2 -3309.838} C_VEL
LIN {X 0,Y 554.494,Z 335.546,A -85,B 0,C 180,E1 -3311.915,E2 -3311.915} C_VEL
LIN {X 0,Y 554.31,Z 350.735,A -85,B 0,C 180,E1 -3312.26,E2 -3312.26} C_VEL
LIN {X 0,Y 554.041,Z 365.745,A -85,B 0,C 180,E1 -3312.752,E2 -3312.752} C_VEL
LIN {X 0,Y 553.727,Z 380.744,A -85,B 0,C 180,E1 -3313.407,E2 -3313.407} C_VEL
LIN {X 0,Y 553.402,Z 394.23,A -85,B 0,C 180,E1 -3314.155,E2 -3314.155} C_VEL
LIN {X 0,Y 553.078,Z 408.145,A -85,B 0,C 180,E1 -3315.103,E2 -3315.103} C_VEL
LIN {X 0,Y 552.76,Z 420.355,A -85,B 0,C 180,E1 -3316.114,E2 -3316.114} C_VEL
LIN {X 0,Y 552.482,Z 432.508,A -85,B 0,C 180,E1 -3317.324,E2 -3317.324} C_VEL
LIN {X 0,Y 552.216,Z 442.483,A -85,B 0,C 180,E1 -3318.513,E2 -3318.513} C_VEL
LIN {X 0,Y 552.124,Z 451.084,A -85,B 0,C 180,E1 -3319.735,E2 -3319.735} C_VEL
LIN {X 0,Y 551.921,Z 458.742,A -85,B 0,C 180,E1 -3321.026,E2 -3321.026} C_VEL
LIN {X 0,Y 551.837,Z 465.089,A -85,B 0,C 180,E1 -3322.315,E2 -3322.315} C_VEL
LIN {X 0,Y 551.769,Z 470.569,A -85,B 0,C 180,E1 -3323.681,E2 -3323.681} C_VEL
LIN {X 0,Y 551.713,Z 474.386,A -85,B 0,C 180,E1 -3324.884,E2 -3324.884} C_VEL
LIN {X 0,Y 551.73,Z 477.887,A -85,B 0,C 180,E1 -3326.348,E2 -3326.348} C_VEL
LIN {X 0,Y 551.655,Z 480.19,A -85,B 0,C 180,E1 -3327.81,E2 -3327.81} C_VEL
LIN {X 0,Y 551.637,Z 481.348,A -85,B 0,C 180,E1 -3329.27,E2 -3329.27} C_VEL
LIN {X 0,Y 551.637,Z 481.347,A -85,B 0,C 180,E1 -3330.73,E2 -3330.73} C_VEL
LIN {X 0,Y 551.655,Z 480.187,A -85,B 0,C 180,E1 -3332.19,E2 -3332.19} C_VEL
LIN {X 0,Y 551.73,Z 477.884,A -85,B 0,C 180,E1 -3333.652,E2 -3333.652} C_VEL
LIN {X 0,Y 551.713,Z 474.387,A -85,B 0,C 180,E1 -3335.116,E2 -3335.116} C_VEL
LIN {X 0,Y 551.82,Z 469.609,A -85,B 0,C 180,E1 -3336.582,E2 -3336.582} C_VEL
LIN {X 0,Y 551.876,Z 463.42,A -85,B 0,C 180,E1 -3338.053,E2 -3338.053} C_VEL
LIN {X 0,Y 551.95,Z 455.643,A -85,B 0,C 180,E1 -3339.528,E2 -3339.528} C_VEL
LIN {X 0,Y 552.183,Z 447.366,A -85,B 0,C 180,E1 -3340.821,E2 -3340.821} C_VEL
LIN {X 0,Y 552.352,Z 437.391,A -85,B 0,C 180,E1 -3342.119,E2 -3342.119} C_VEL
LIN {X 0,Y 552.609,Z 427.184,A -85,B 0,C 180,E1 -3343.234,E2 -3343.234} C_VEL
LIN {X 0,Y 552.907,Z 415.018,A -85,B 0,C 180,E1 -3344.351,E2 -3344.351} C_VEL
LIN {X 0,Y 553.243,Z 402.428,A -85,B 0,C 180,E1 -3345.31,E2 -3345.31} C_VEL
LIN {X 0,Y 553.509,Z 389.475,A -85,B 0,C 180,E1 -3346.126,E2 -3346.126} C_VEL
LIN {X 0,Y 553.863,Z 374.776,A -85,B 0,C 180,E1 -3346.874,E2 -3346.874} C_VEL
LIN {X 0,Y 554.141,Z 360.557,A -85,B 0,C 180,E1 -3347.435,E2 -3347.435} C_VEL
LIN {X 0,Y 554.355,Z 346.555,A -85,B 0,C 180,E1 -3347.848,E2 -3347.848} C_VEL
LIN {X 0,Y 554.525,Z 331.022,A -85,B 0,C 180,E1 -3348.156,E2 -3348.156} C_VEL
LIN {X 0,Y 555.142,Z 180.296,A -85,B 0,C 180,E1 -3350.163,E2 -3350.163} C_VEL
LIN {X 0,Y 553.278,Z 170.077,A -85,B 0,C 180,E1 -3350.396,E2 -3350.396} C_VEL
LIN {X 0,Y 553.593,Z 150.099,A -85,B 0,C 180,E1 -3352.978,E2 -3352.978} C_VEL
LIN {X 0,Y 553.861,Z 135.227,A -85,B 0,C 180,E1 -3354.944,E2 -3354.944} C_VEL
LIN {X 0,Y 552.15,Z 127.412,A -85,B 0,C 180,E1 -3356.125,E2 -3356.125} C_VEL
LIN {X 0,Y 552.111,Z 127.334,A -85,B 0,C 180,E1 -3358.928,E2 -3358.928} C_VEL
LIN {X 0,Y 552.112,Z 127.328,A -85,B 0,C 180,E1 -3361.476,E2 -3361.476} C_VEL
LIN {X 0,Y 552.133,Z 127.338,A -85,B 0,C 180,E1 -3364.17,E2 -3364.17} C_VEL
LIN {X 0,Y 552.106,Z 127.333,A -85,B 0,C 180,E1 -3366.747,E2 -3366.747} C_VEL
LIN {X 0,Y 552.134,Z 127.331,A -85,B 0,C 180,E1 -3369.527,E2 -3369.527} C_VEL
LIN {X 0,Y 552.13,Z 127.33,A -85,B 0,C 180,E1 -3372.426,E2 -3372.426} C_VEL
LIN {X 0,Y 552.097,Z 127.338,A -85,B 0,C 180,E1 -3375.563,E2 -3375.563} C_VEL
LIN {X 0,Y 552.122,Z 127.327,A -85,B 0,C 180,E1 -3378.554,E2 -3378.554} C_VEL
LIN {X 0,Y 552.118,Z 127.334,A -85,B 0,C 180,E1 -3381.411,E2 -3381.411} C_VEL
LIN {X 0,Y 552.086,Z 127.334,A -85,B 0,C 180,E1 -3384.156,E2 -3384.156} C_VEL
LIN {X 0,Y 552.107,Z 127.325,A -85,B 0,C 180,E1 -3386.814,E2 -3386.814} C_VEL
LIN {X 0,Y 552.1,Z 127.338,A -85,B 0,C 180,E1 -3389.391,E2 -3389.391} C_VEL
LIN {X 0,Y 552.107,Z 127.333,A -85,B 0,C 180,E1 -3391.902,E2 -3391.902} C_VEL
LIN {X 0,Y 552.139,Z 127.327,A -85,B 0,C 180,E1 -3394.654,E2 -3394.654} C_VEL
LIN {X 0,Y 552.092,Z 127.336,A -85,B 0,C 180,E1 -3397.549,E2 -3397.549} C_VEL
LIN {X 0,Y 552.146,Z 127.327,A -85,B 0,C 180,E1 -3400.375,E2 -3400.375} C_VEL
LIN {X 0,Y 552.124,Z 127.337,A -85,B 0,C 180,E1 -3402.976,E2 -3402.976} C_VEL
LIN {X 0,Y 552.124,Z 127.329,A -85,B 0,C 180,E1 -3406.004,E2 -3406.004} C_VEL
LIN {X 0,Y 552.162,Z 127.329,A -85,B 0,C 180,E1 -3408.993,E2 -3408.993} C_VEL
LIN {X 0,Y 552.151,Z 127.326,A -85,B 0,C 180,E1 -3411.952,E2 -3411.952} C_VEL
LIN {X 0,Y 552.223,Z 127.32,A -85,B 0,C 180,E1 -3414.889,E2 -3414.889} C_VEL
LIN {X 0,Y 552.225,Z 127.316,A -85,B 0,C 180,E1 -3417.812,E2 -3417.812} C_VEL
LIN {X 0,Y 552.24,Z 127.318,A -85,B 0,C 180,E1 -3420.729,E2 -3420.729} C_VEL
LIN {X 0,Y 552.191,Z 127.322,A -85,B 0,C 180,E1 -3422.918,E2 -3422.918} C_VEL
LIN {X 0,Y 552.193,Z 127.324,A -85,B 0,C 180,E1 -3425.844,E2 -3425.844} C_VEL
LIN {X 0,Y 552.15,Z 127.326,A -85,B 0,C 180,E1 -3428.786,E2 -3428.786} C_VEL
LIN {X 0,Y 552.163,Z 127.329,A -85,B 0,C 180,E1 -3431.751,E2 -3431.751} C_VEL
LIN {X 0,Y 552.13,Z 127.328,A -85,B 0,C 180,E1 -3434.749,E2 -3434.749} C_VEL
LIN {X 0,Y 552.081,Z 127.342,A -85,B 0,C 180,E1 -3437.79,E2 -3437.79} C_VEL
LIN {X 0,Y 552.125,Z 127.335,A -85,B 0,C 180,E1 -3440.102,E2 -3440.102} C_VEL
LIN {X 0,Y 552.085,Z 127.337,A -85,B 0,C 180,E1 -3442.451,E2 -3442.451} C_VEL
LIN {X 0,Y 552.085,Z 127.335,A -85,B 0,C 180,E1 -3445.334,E2 -3445.334} C_VEL
LIN {X 0,Y 552.064,Z 127.341,A -85,B 0,C 180,E1 -3448.101,E2 -3448.101} C_VEL
LIN {X 0,Y 552.093,Z 127.329,A -85,B 0,C 180,E1 -3450.61,E2 -3450.61} C_VEL
LIN {X 0,Y 552.104,Z 127.326,A -85,B 0,C 180,E1 -3453.187,E2 -3453.187} C_VEL
LIN {X 0,Y 552.086,Z 127.331,A -85,B 0,C 180,E1 -3453.778,E2 -3453.778} C_VEL
LIN {X 0,Y 551.445,Z 127.417,A -85,B 0,C 180,E1 -3454.386,E2 -3454.386} C_VEL
LIN {X 0,Y 548.631,Z 127.77,A -85,B 0,C 180,E1 -3455.375,E2 -3455.375} C_VEL
LIN {X 0,Y 546.222,Z 128.067,A -85,B 0,C 180,E1 -3456.17,E2 -3456.17} C_VEL
LIN {X 0,Y 545.159,Z 128.199,A -85,B 0,C 180,E1 -3456.784,E2 -3456.784} C_VEL
LIN {X 0,Y 545.057,Z 128.214,A -85,B 0,C 180,E1 -3456.992,E2 -3456.992} C_VEL
LIN {X 0,Y 545.062,Z 128.201,A -85,B 0,C 180,E1 -3460.143,E2 -3460.143} C_VEL
LIN {X 0,Y 545.018,Z 128.221,A -85,B 0,C 180,E1 -3463.113,E2 -3463.113} C_VEL
LIN {X 0,Y 545.028,Z 128.21,A -85,B 0,C 180,E1 -3466.229,E2 -3466.229} C_VEL
LIN {X 0,Y 545.028,Z 128.22,A -85,B 0,C 180,E1 -3468.88,E2 -3468.88} C_VEL
LIN {X 0,Y 545.046,Z 128.214,A -85,B 0,C 180,E1 -3471.762,E2 -3471.762} C_VEL
LIN {X 0,Y 545.022,Z 128.217,A -85,B 0,C 180,E1 -3474.53,E2 -3474.53} C_VEL
LIN {X 0,Y 545.061,Z 128.216,A -85,B 0,C 180,E1 -3477.211,E2 -3477.211} C_VEL
LIN {X 0,Y 545.018,Z 128.207,A -85,B 0,C 180,E1 -3479.808,E2 -3479.808} C_VEL
LIN {X 0,Y 545.023,Z 128.213,A -85,B 0,C 180,E1 -3482.842,E2 -3482.842} C_VEL
LIN {X 0,Y 545.076,Z 128.416,A -85,B 0,C 180,E1 -3484.741,E2 -3484.741} C_VEL
LIN {X 0,Y 546.848,Z 136.67,A -85,B 0,C 180,E1 -3486.036,E2 -3486.036} C_VEL
LIN {X 0,Y 546.502,Z 152.821,A -85,B 0,C 180,E1 -3488.301,E2 -3488.301} C_VEL
LIN {X 0,Y 546.348,Z 160.889,A -85,B 0,C 180,E1 -3489.389,E2 -3489.389} C_VEL
LIN {X 0,Y 548.519,Z 171.665,A -85,B 0,C 180,E1 -3489.642,E2 -3489.642} C_VEL
LIN {X 0,Y 547.726,Z 326.488,A -85,B 0,C 180,E1 -3491.741,E2 -3491.741} C_VEL
LIN {X 0,Y 547.533,Z 341.962,A -85,B 0,C 180,E1 -3492.106,E2 -3492.106} C_VEL
LIN {X 0,Y 547.25,Z 357.24,A -85,B 0,C 180,E1 -3492.627,E2 -3492.627} C_VEL
LIN {X 0,Y 546.908,Z 371.868,A -85,B 0,C 180,E1 -3493.29,E2 -3493.29} C_VEL
LIN {X 0,Y 546.507,Z 385.173,A -85,B 0,C 180,E1 -3494.045,E2 -3494.045} C_VEL
LIN {X 0,Y 546.179,Z 398.372,A -85,B 0,C 180,E1 -3494.966,E2 -3494.966} C_VEL
LIN {X 0,Y 545.79,Z 410.965,A -85,B 0,C 180,E1 -3496.029,E2 -3496.029} C_VEL
LIN {X 0,Y 545.526,Z 422.136,A -85,B 0,C 180,E1 -3497.16,E2 -3497.16} C_VEL
LIN {X 0,Y 545.229,Z 432.572,A -85,B 0,C 180,E1 -3498.419,E2 -3498.419} C_VEL
LIN {X 0,Y 545.05,Z 442.012,A -85,B 0,C 180,E1 -3499.788,E2 -3499.788} C_VEL
LIN {X 0,Y 544.846,Z 449.5,A -85,B 0,C 180,E1 -3501.095,E2 -3501.095} C_VEL
LIN {X 0,Y 544.746,Z 456.506,A -85,B 0,C 180,E1 -3502.587,E2 -3502.587} C_VEL
LIN {X 0,Y 544.708,Z 462.015,A -85,B 0,C 180,E1 -3504.075,E2 -3504.075} C_VEL
LIN {X 0,Y 544.605,Z 466.18,A -85,B 0,C 180,E1 -3505.559,E2 -3505.559} C_VEL
LIN {X 0,Y 544.643,Z 469.111,A -85,B 0,C 180,E1 -3507.041,E2 -3507.041} C_VEL
LIN {X 0,Y 544.543,Z 470.878,A -85,B 0,C 180,E1 -3508.521,E2 -3508.521} C_VEL
LIN {X 0,Y 544.539,Z 471.496,A -85,B 0,C 180,E1 -3510,E2 -3510} C_VEL
LIN {X 0,Y 544.544,Z 470.938,A -85,B 0,C 180,E1 -3511.479,E2 -3511.479} C_VEL
LIN {X 0,Y 544.645,Z 469.252,A -85,B 0,C 180,E1 -3512.959,E2 -3512.959} C_VEL
LIN {X 0,Y 544.605,Z 466.399,A -85,B 0,C 180,E1 -3514.441,E2 -3514.441} C_VEL
LIN {X 0,Y 544.696,Z 462.312,A -85,B 0,C 180,E1 -3515.925,E2 -3515.925} C_VEL
LIN {X 0,Y 544.746,Z 456.894,A -85,B 0,C 180,E1 -3517.413,E2 -3517.413} C_VEL
LIN {X 0,Y 544.846,Z 449.991,A -85,B 0,C 180,E1 -3518.905,E2 -3518.905} C_VEL
LIN {X 0,Y 545.081,Z 441.378,A -85,B 0,C 180,E1 -3520.399,E2 -3520.399} C_VEL
LIN {X 0,Y 545.227,Z 432.113,A -85,B 0,C 180,E1 -3521.73,E2 -3521.73} C_VEL
LIN {X 0,Y 545.486,Z 422.93,A -85,B 0,C 180,E1 -3522.841,E2 -3522.841} C_VEL
LIN {X 0,Y 545.818,Z 410.905,A -85,B 0,C 180,E1 -3524.066,E2 -3524.066} C_VEL
LIN {X 0,Y 546.172,Z 398.918,A -85,B 0,C 180,E1 -3525.08,E2 -3525.08} C_VEL
LIN {X 0,Y 546.552,Z 385.082,A -85,B 0,C 180,E1 -3526.049,E2 -3526.049} C_VEL
LIN {X 0,Y 546.912,Z 371.762,A -85,B 0,C 180,E1 -3526.806,E2 -3526.806} C_VEL
LIN {X 0,Y 547.273,Z 357.077,A -85,B 0,C 180,E1 -3527.468,E2 -3527.468} C_VEL
LIN {X 0,Y 547.564,Z 341.985,A -85,B 0,C 180,E1 -3527.982,E2 -3527.982} C_VEL
LIN {X 0,Y 547.762,Z 326.928,A -85,B 0,C 180,E1 -3528.338,E2 -3528.338} C_VEL
LIN {X 0,Y 548.114,Z 256.653,A -85,B 0,C 180,E1 -3529.304,E2 -3529.304} C_VEL
LIN {X 0,Y 548.395,Z 170.669,A -85,B 0,C 180,E1 -3530.466,E2 -3530.466} C_VEL
LIN {X 0,Y 546.331,Z 160.911,A -85,B 0,C 180,E1 -3530.7,E2 -3530.7} C_VEL
LIN {X 0,Y 546.811,Z 142.133,A -85,B 0,C 180,E1 -3533.28,E2 -3533.28} C_VEL
LIN {X 0,Y 546.772,Z 136.147,A -85,B 0,C 180,E1 -3534.132,E2 -3534.132} C_VEL
LIN {X 0,Y 545.047,Z 128.363,A -85,B 0,C 180,E1 -3535.375,E2 -3535.375} C_VEL
LIN {X 0,Y 544.997,Z 128.221,A -85,B 0,C 180,E1 -3537.661,E2 -3537.661} C_VEL
LIN {X 0,Y 545.02,Z 128.206,A -85,B 0,C 180,E1 -3540.236,E2 -3540.236} C_VEL
LIN {X 0,Y 545.062,Z 128.218,A -85,B 0,C 180,E1 -3543.059,E2 -3543.059} C_VEL
LIN {X 0,Y 545.017,Z 128.216,A -85,B 0,C 180,E1 -3545.67,E2 -3545.67} C_VEL
LIN {X 0,Y 545.044,Z 128.214,A -85,B 0,C 180,E1 -3548.238,E2 -3548.238} C_VEL
LIN {X 0,Y 545.015,Z 128.223,A -85,B 0,C 180,E1 -3551.121,E2 -3551.121} C_VEL
LIN {X 0,Y 545.031,Z 128.21,A -85,B 0,C 180,E1 -3554.132,E2 -3554.132} C_VEL
LIN {X 0,Y 545.018,Z 128.223,A -85,B 0,C 180,E1 -3556.887,E2 -3556.887} C_VEL
LIN {X 0,Y 545.051,Z 128.203,A -85,B 0,C 180,E1 -3559.856,E2 -3559.856} C_VEL
LIN {X 0,Y 545.065,Z 128.213,A -85,B 0,C 180,E1 -3563.075,E2 -3563.075} C_VEL
LIN {X 0,Y 545.047,Z 128.215,A -85,B 0,C 180,E1 -3566.327,E2 -3566.327} C_VEL
LIN {X 0,Y 545.055,Z 128.207,A -85,B 0,C 180,E1 -3568.951,E2 -3568.951} C_VEL
LIN {X 0,Y 545.04,Z 128.212,A -85,B 0,C 180,E1 -3571.504,E2 -3571.504} C_VEL
LIN {X 0,Y 545.045,Z 128.216,A -85,B 0,C 180,E1 -3573.998,E2 -3573.998} C_VEL
LIN {X 0,Y 545.072,Z 128.215,A -85,B 0,C 180,E1 -3576.44,E2 -3576.44} C_VEL
LIN {X 0,Y 545.086,Z 128.207,A -85,B 0,C 180,E1 -3579.627,E2 -3579.627} C_VEL
LIN {X 0,Y 545.031,Z 128.214,A -85,B 0,C 180,E1 -3582.748,E2 -3582.748} C_VEL
LIN {X 0,Y 545.082,Z 128.211,A -85,B 0,C 180,E1 -3585.82,E2 -3585.82} C_VEL
LIN {X 0,Y 545.119,Z 128.203,A -85,B 0,C 180,E1 -3588.849,E2 -3588.849} C_VEL
LIN {X 0,Y 545.095,Z 128.21,A -85,B 0,C 180,E1 -3591.846,E2 -3591.846} C_VEL
LIN {X 0,Y 545.196,Z 128.193,A -85,B 0,C 180,E1 -3594.823,E2 -3594.823} C_VEL
LIN {X 0,Y 545.197,Z 128.197,A -85,B 0,C 180,E1 -3597.784,E2 -3597.784} C_VEL
LIN {X 0,Y 545.205,Z 128.192,A -85,B 0,C 180,E1 -3600.739,E2 -3600.739} C_VEL
LIN {X 0,Y 545.163,Z 128.197,A -85,B 0,C 180,E1 -3602.956,E2 -3602.956} C_VEL
LIN {X 0,Y 545.17,Z 128.198,A -85,B 0,C 180,E1 -3605.919,E2 -3605.919} C_VEL
LIN {X 0,Y 545.102,Z 128.207,A -85,B 0,C 180,E1 -3608.9,E2 -3608.9} C_VEL
LIN {X 0,Y 545.107,Z 128.205,A -85,B 0,C 180,E1 -3611.905,E2 -3611.905} C_VEL
LIN {X 0,Y 545.084,Z 128.213,A -85,B 0,C 180,E1 -3614.944,E2 -3614.944} C_VEL
LIN {X 0,Y 545.06,Z 128.21,A -85,B 0,C 180,E1 -3618.026,E2 -3618.026} C_VEL
LIN {X 0,Y 545.093,Z 128.206,A -85,B 0,C 180,E1 -3620.372,E2 -3620.372} C_VEL
LIN {X 0,Y 545.075,Z 128.209,A -85,B 0,C 180,E1 -3623.56,E2 -3623.56} C_VEL
LIN {X 0,Y 545.071,Z 128.206,A -85,B 0,C 180,E1 -3626.001,E2 -3626.001} C_VEL
LIN {X 0,Y 545.09,Z 128.215,A -85,B 0,C 180,E1 -3628.748,E2 -3628.748} C_VEL
LIN {X 0,Y 545.056,Z 128.205,A -85,B 0,C 180,E1 -3631.915,E2 -3631.915} C_VEL
LIN {X 0,Y 545.06,Z 128.211,A -85,B 0,C 180,E1 -3634.565,E2 -3634.565} C_VEL
LIN {X 0,Y 545.037,Z 128.213,A -85,B 0,C 180,E1 -3637.304,E2 -3637.304} C_VEL
LIN {X 0,Y 545.066,Z 128.21,A -85,B 0,C 180,E1 -3640.142,E2 -3640.142} C_VEL
LIN {X 0,Y 545.08,Z 128.209,A -85,B 0,C 180,E1 -3643.106,E2 -3643.106} C_VEL
LIN {X 0,Y 545.05,Z 128.214,A -85,B 0,C 180,E1 -3646.226,E2 -3646.226} C_VEL
LIN {X 0,Y 545.083,Z 128.208,A -85,B 0,C 180,E1 -3648.885,E2 -3648.885} C_VEL
LIN {X 0,Y 545.085,Z 128.206,A -85,B 0,C 180,E1 -3650.819,E2 -3650.819} C_VEL
LIN {X 0,Y 545.043,Z 128.217,A -85,B 0,C 180,E1 -3653.62,E2 -3653.62} C_VEL
LIN {X 0,Y 545.067,Z 128.21,A -85,B 0,C 180,E1 -3656.328,E2 -3656.328} C_VEL
LIN {X 0,Y 545.067,Z 128.206,A -85,B 0,C 180,E1 -3658.952,E2 -3658.952} C_VEL
LIN {X 0,Y 545.102,Z 128.202,A -85,B 0,C 180,E1 -3661.508,E2 -3661.508} C_VEL
LIN {X 0,Y 545.114,Z 128.423,A -85,B 0,C 180,E1 -3663.692,E2 -3663.692} C_VEL
LIN {X 0,Y 546.957,Z 136.576,A -85,B 0,C 180,E1 -3664.911,E2 -3664.911} C_VEL
LIN {X 0,Y 546.946,Z 144.272,A -85,B 0,C 180,E1 -3665.951,E2 -3665.951} C_VEL
LIN {X 0,Y 546.439,Z 164.988,A -85,B 0,C 180,E1 -3668.695,E2 -3668.695} C_VEL
LIN {X 0,Y 546.411,Z 170.246,A -85,B 0,C 180,E1 -3669.35,E2 -3669.35} C_VEL
LIN {X 0,Y 548.5,Z 181.407,A -85,B 0,C 180,E1 -3669.598,E2 -3669.598} C_VEL
LIN {X 0,Y 547.748,Z 335.363,A -85,B 0,C 180,E1 -3671.682,E2 -3671.682} C_VEL
LIN {X 0,Y 547.552,Z 350.808,A -85,B 0,C 180,E1 -3672.037,E2 -3672.037} C_VEL
LIN {X 0,Y 547.256,Z 365.679,A -85,B 0,C 180,E1 -3672.531,E2 -3672.531} C_VEL
LIN {X 0,Y 546.935,Z 378.689,A -85,B 0,C 180,E1 -3673.098,E2 -3673.098} C_VEL
LIN {X 0,Y 546.568,Z 392.58,A -85,B 0,C 180,E1 -3673.855,E2 -3673.855} C_VEL
LIN {X 0,Y 546.285,Z 404.535,A -85,B 0,C 180,E1 -3674.651,E2 -3674.651} C_VEL
LIN {X 0,Y 545.915,Z 417.094,A -85,B 0,C 180,E1 -3675.651,E2 -3675.651} C_VEL
LIN {X 0,Y 545.586,Z 428.931,A -85,B 0,C 180,E1 -3676.782,E2 -3676.782} C_VEL
LIN {X 0,Y 545.315,Z 438.89,A -85,B 0,C 180,E1 -3677.911,E2 -3677.911} C_VEL
LIN {X 0,Y 545.155,Z 447.366,A -85,B 0,C 180,E1 -3679.038,E2 -3679.038} C_VEL
LIN {X 0,Y 544.904,Z 455.647,A -85,B 0,C 180,E1 -3680.348,E2 -3680.348} C_VEL
LIN {X 0,Y 544.818,Z 463.422,A -85,B 0,C 180,E1 -3681.842,E2 -3681.842} C_VEL
LIN {X 0,Y 544.704,Z 470.08,A -85,B 0,C 180,E1 -3683.456,E2 -3683.456} C_VEL
LIN {X 0,Y 544.642,Z 474.386,A -85,B 0,C 180,E1 -3684.818,E2 -3684.818} C_VEL
LIN {X 0,Y 544.645,Z 477.887,A -85,B 0,C 180,E1 -3686.301,E2 -3686.301} C_VEL
LIN {X 0,Y 544.569,Z 480.189,A -85,B 0,C 180,E1 -3687.781,E2 -3687.781} C_VEL
LIN {X 0,Y 544.537,Z 481.348,A -85,B 0,C 180,E1 -3689.26,E2 -3689.26} C_VEL
LIN {X 0,Y 544.537,Z 481.347,A -85,B 0,C 180,E1 -3690.739,E2 -3690.739} C_VEL
LIN {X 0,Y 544.569,Z 480.186,A -85,B 0,C 180,E1 -3692.219,E2 -3692.219} C_VEL
LIN {X 0,Y 544.645,Z 477.883,A -85,B 0,C 180,E1 -3693.699,E2 -3693.699} C_VEL
LIN {X 0,Y 544.642,Z 474.386,A -85,B 0,C 180,E1 -3695.182,E2 -3695.182} C_VEL
LIN {X 0,Y 544.752,Z 469.609,A -85,B 0,C 180,E1 -3696.668,E2 -3696.668} C_VEL
LIN {X 0,Y 544.818,Z 463.419,A -85,B 0,C 180,E1 -3698.158,E2 -3698.158} C_VEL
LIN {X 0,Y 544.904,Z 455.642,A -85,B 0,C 180,E1 -3699.652,E2 -3699.652} C_VEL
LIN {X 0,Y 545.149,Z 447.366,A -85,B 0,C 180,E1 -3700.962,E2 -3700.962} C_VEL
LIN {X 0,Y 545.357,Z 437.375,A -85,B 0,C 180,E1 -3702.277,E2 -3702.277} C_VEL
LIN {X 0,Y 545.639,Z 427.148,A -85,B 0,C 180,E1 -3703.406,E2 -3703.406} C_VEL
LIN {X 0,Y 545.974,Z 414.961,A -85,B 0,C 180,E1 -3704.537,E2 -3704.537} C_VEL
LIN {X 0,Y 546.376,Z 401.304,A -85,B 0,C 180,E1 -3705.582,E2 -3705.582} C_VEL
LIN {X 0,Y 546.743,Z 387.785,A -85,B 0,C 180,E1 -3706.427,E2 -3706.427} C_VEL
LIN {X 0,Y 547.046,Z 373.689,A -85,B 0,C 180,E1 -3707.138,E2 -3707.138} C_VEL
LIN {X 0,Y 547.373,Z 359.182,A -85,B 0,C 180,E1 -3707.706,E2 -3707.706} C_VEL
LIN {X 0,Y 547.613,Z 344.076,A -85,B 0,C 180,E1 -3708.139,E2 -3708.139} C_VEL
LIN {X 0,Y 547.819,Z 328.274,A -85,B 0,C 180,E1 -3708.429,E2 -3708.429} C_VEL
LIN {X 0,Y 548.5,Z 181.412,A -85,B 0,C 180,E1 -3710.402,E2 -3710.402} C_VEL
LIN {X 0,Y 546.408,Z 170.207,A -85,B 0,C 180,E1 -3710.652,E2 -3710.652} C_VEL
LIN {X 0,Y 546.774,Z 150.038,A -85,B 0,C 180,E1 -3713.281,E2 -3713.281} C_VEL
LIN {X 0,Y 547.137,Z 138.074,A -85,B 0,C 180,E1 -3714.877,E2 -3714.877} C_VEL
LIN {X 0,Y 545.107,Z 128.331,A -85,B 0,C 180,E1 -3716.334,E2 -3716.334} C_VEL
LIN {X 0,Y 545.065,Z 128.212,A -85,B 0,C 180,E1 -3719.338,E2 -3719.338} C_VEL
LIN {X 0,Y 545.056,Z 128.204,A -85,B 0,C 180,E1 -3721.915,E2 -3721.915} C_VEL
LIN {X 0,Y 545.063,Z 128.213,A -85,B 0,C 180,E1 -3724.565,E2 -3724.565} C_VEL
LIN {X 0,Y 545.037,Z 128.214,A -85,B 0,C 180,E1 -3727.304,E2 -3727.304} C_VEL
LIN {X 0,Y 545.069,Z 128.215,A -85,B 0,C 180,E1 -3730.142,E2 -3730.142} C_VEL
LIN {X 0,Y 545.079,Z 128.207,A -85,B 0,C 180,E1 -3733.107,E2 -3733.107} C_VEL
LIN {X 0,Y 545.068,Z 128.212,A -85,B 0,C 180,E1 -3736.224,E2 -3736.224} C_VEL
LIN {X 0,Y 545.082,Z 128.204,A -85,B 0,C 180,E1 -3738.886,E2 -3738.886} C_VEL
LIN {X 0,Y 545.053,Z 128.218,A -85,B 0,C 180,E1 -3741.763,E2 -3741.763} C_VEL
LIN {X 0,Y 545.037,Z 128.211,A -85,B 0,C 180,E1 -3744.532,E2 -3744.532} C_VEL
LIN {X 0,Y 545.065,Z 128.203,A -85,B 0,C 180,E1 -3747.211,E2 -3747.211} C_VEL
LIN {X 0,Y 545.062,Z 128.212,A -85,B 0,C 180,E1 -3749.81,E2 -3749.81} C_VEL
LIN {X 0,Y 545.079,Z 128.208,A -85,B 0,C 180,E1 -3752.344,E2 -3752.344} C_VEL
LIN {X 0,Y 545.107,Z 128.205,A -85,B 0,C 180,E1 -3754.82,E2 -3754.82} C_VEL
LIN {X 0,Y 545.037,Z 128.219,A -85,B 0,C 180,E1 -3757.242,E2 -3757.242} C_VEL
LIN {X 0,Y 545.118,Z 128.203,A -85,B 0,C 180,E1 -3760.415,E2 -3760.415} C_VEL
LIN {X 0,Y 545.056,Z 128.209,A -85,B 0,C 180,E1 -3763.521,E2 -3763.521} C_VEL
LIN {X 0,Y 545.086,Z 128.206,A -85,B 0,C 180,E1 -3765.82,E2 -3765.82} C_VEL
LIN {X 0,Y 545.119,Z 128.208,A -85,B 0,C 180,E1 -3768.849,E2 -3768.849} C_VEL
LIN {X 0,Y 545.099,Z 128.204,A -85,B 0,C 180,E1 -3771.847,E2 -3771.847} C_VEL
LIN {X 0,Y 545.2,Z 128.196,A -85,B 0,C 180,E1 -3774.823,E2 -3774.823} C_VEL
LIN {X 0,Y 545.196,Z 128.191,A -85,B 0,C 180,E1 -3777.784,E2 -3777.784} C_VEL
LIN {X 0,Y 545.21,Z 128.194,A -85,B 0,C 180,E1 -3780.739,E2 -3780.739} C_VEL
LIN {X 0,Y 545.158,Z 128.197,A -85,B 0,C 180,E1 -3782.956,E2 -3782.956} C_VEL
LIN {X 0,Y 545.165,Z 128.2,A -85,B 0,C 180,E1 -3785.92,E2 -3785.92} C_VEL
LIN {X 0,Y 545.107,Z 128.202,A -85,B 0,C 180,E1 -3788.9,E2 -3788.9} C_VEL
LIN {X 0,Y 545.106,Z 128.21,A -85,B 0,C 180,E1 -3791.905,E2 -3791.905} C_VEL
LIN {X 0,Y 545.082,Z 128.204,A -85,B 0,C 180,E1 -3794.944,E2 -3794.944} C_VEL
LIN {X 0,Y 545.051,Z 128.219,A -85,B 0,C 180,E1 -3798.027,E2 -3798.027} C_VEL
LIN {X 0,Y 545.091,Z 128.207,A -85,B 0,C 180,E1 -3800.372,E2 -3800.372} C_VEL
LIN {X 0,Y 545.073,Z 128.214,A -85,B 0,C 180,E1 -3803.56,E2 -3803.56} C_VEL
LIN {X 0,Y 545.058,Z 128.21,A -85,B 0,C 180,E1 -3806.827,E2 -3806.827} C_VEL
LIN {X 0,Y 545.029,Z 128.218,A -85,B 0,C 180,E1 -3809.341,E2 -3809.341} C_VEL
LIN {X 0,Y 545.053,Z 128.203,A -85,B 0,C 180,E1 -3811.915,E2 -3811.915} C_VEL
LIN {X 0,Y 545.047,Z 128.209,A -85,B 0,C 180,E1 -3814.566,E2 -3814.566} C_VEL
LIN {X 0,Y 545.057,Z 128.214,A -85,B 0,C 180,E1 -3816.992,E2 -3816.992} C_VEL
LIN {X 0,Y 544.35,Z 128.306,A -85,B 0,C 180,E1 -3817.608,E2 -3817.608} C_VEL
LIN {X 0,Y 541.485,Z 128.658,A -85,B 0,C 180,E1 -3818.609,E2 -3818.609} C_VEL
LIN {X 0,Y 539.092,Z 128.951,A -85,B 0,C 180,E1 -3819.415,E2 -3819.415} C_VEL
LIN {X 0,Y 538.07,Z 129.072,A -85,B 0,C 180,E1 -3820.037,E2 -3820.037} C_VEL
LIN {X 0,Y 537.989,Z 129.081,A -85,B 0,C 180,E1 -3820.248,E2 -3820.248} C_VEL
LIN {X 0,Y 537.971,Z 129.097,A -85,B 0,C 180,E1 -3822.981,E2 -3822.981} C_VEL
LIN {X 0,Y 538.002,Z 129.085,A -85,B 0,C 180,E1 -3825.929,E2 -3825.929} C_VEL
LIN {X 0,Y 538.006,Z 129.092,A -85,B 0,C 180,E1 -3829.258,E2 -3829.258} C_VEL
LIN {X 0,Y 537.987,Z 129.092,A -85,B 0,C 180,E1 -3832.122,E2 -3832.122} C_VEL
LIN {X 0,Y 537.985,Z 129.099,A -85,B 0,C 180,E1 -3834.915,E2 -3834.915} C_VEL
LIN {X 0,Y 538.01,Z 129.091,A -85,B 0,C 180,E1 -3837.617,E2 -3837.617} C_VEL
LIN {X 0,Y 537.972,Z 129.085,A -85,B 0,C 180,E1 -3840.236,E2 -3840.236} C_VEL
LIN {X 0,Y 537.993,Z 129.088,A -85,B 0,C 180,E1 -3842.792,E2 -3842.792} C_VEL
LIN {X 0,Y 538.011,Z 129.197,A -85,B 0,C 180,E1 -3844.464,E2 -3844.464} C_VEL
LIN {X 0,Y 538.558,Z 131.668,A -85,B 0,C 180,E1 -3844.905,E2 -3844.905} C_VEL
LIN {X 0,Y 540.029,Z 138.988,A -85,B 0,C 180,E1 -3846.04,E2 -3846.04} C_VEL
LIN {X 0,Y 539.535,Z 157.137,A -85,B 0,C 180,E1 -3848.609,E2 -3848.609} C_VEL
LIN {X 0,Y 539.505,Z 161.141,A -85,B 0,C 180,E1 -3849.126,E2 -3849.126} C_VEL
LIN {X 0,Y 541.837,Z 172.207,A -85,B 0,C 180,E1 -3849.386,E2 -3849.386} C_VEL
LIN {X 0,Y 541.005,Z 326.584,A -85,B 0,C 180,E1 -3851.506,E2 -3851.506} C_VEL
LIN {X 0,Y 540.807,Z 342.048,A -85,B 0,C 180,E1 -3851.876,E2 -3851.876} C_VEL
LIN {X 0,Y 540.471,Z 357.321,A -85,B 0,C 180,E1 -3852.402,E2 -3852.402} C_VEL
LIN {X 0,Y 540.089,Z 371.946,A -85,B 0,C 180,E1 -3853.073,E2 -3853.073} C_VEL
LIN {X 0,Y 539.66,Z 385.249,A -85,B 0,C 180,E1 -3853.837,E2 -3853.837} C_VEL
LIN {X 0,Y 539.271,Z 399.091,A -85,B 0,C 180,E1 -3854.821,E2 -3854.821} C_VEL
LIN {X 0,Y 538.855,Z 411.038,A -85,B 0,C 180,E1 -3855.845,E2 -3855.845} C_VEL
LIN {X 0,Y 538.568,Z 422.208,A -85,B 0,C 180,E1 -3856.991,E2 -3856.991} C_VEL
LIN {X 0,Y 538.218,Z 433.151,A -85,B 0,C 180,E1 -3858.335,E2 -3858.335} C_VEL
LIN {X 0,Y 538.021,Z 442.074,A -85,B 0,C 180,E1 -3859.653,E2 -3859.653} C_VEL
LIN {X 0,Y 537.8,Z 449.544,A -85,B 0,C 180,E1 -3860.978,E2 -3860.978} C_VEL
LIN {X 0,Y 537.663,Z 456.531,A -85,B 0,C 180,E1 -3862.489,E2 -3862.489} C_VEL
LIN {X 0,Y 537.62,Z 462.025,A -85,B 0,C 180,E1 -3863.997,E2 -3863.997} C_VEL
LIN {X 0,Y 537.507,Z 466.18,A -85,B 0,C 180,E1 -3865.5,E2 -3865.5} C_VEL
LIN {X 0,Y 537.543,Z 469.11,A -85,B 0,C 180,E1 -3867.002,E2 -3867.002} C_VEL
LIN {X 0,Y 537.448,Z 470.877,A -85,B 0,C 180,E1 -3868.501,E2 -3868.501} C_VEL
LIN {X 0,Y 537.44,Z 471.496,A -85,B 0,C 180,E1 -3870,E2 -3870} C_VEL
LIN {X 0,Y 537.449,Z 470.937,A -85,B 0,C 180,E1 -3871.499,E2 -3871.499} C_VEL
LIN {X 0,Y 537.545,Z 469.25,A -85,B 0,C 180,E1 -3872.998,E2 -3872.998} C_VEL
LIN {X 0,Y 537.507,Z 466.397,A -85,B 0,C 180,E1 -3874.5,E2 -3874.5} C_VEL
LIN {X 0,Y 537.594,Z 462.317,A -85,B 0,C 180,E1 -3876.003,E2 -3876.003} C_VEL
LIN {X 0,Y 537.662,Z 456.913,A -85,B 0,C 180,E1 -3877.511,E2 -3877.511} C_VEL
LIN {X 0,Y 537.797,Z 450.028,A -85,B 0,C 180,E1 -3879.022,E2 -3879.022} C_VEL
LIN {X 0,Y 538.037,Z 441.434,A -85,B 0,C 180,E1 -3880.537,E2 -3880.537} C_VEL
LIN {X 0,Y 538.238,Z 431.981,A -85,B 0,C 180,E1 -3881.909,E2 -3881.909} C_VEL
LIN {X 0,Y 538.567,Z 421.266,A -85,B 0,C 180,E1 -3883.201,E2 -3883.201} C_VEL
LIN {X 0,Y 538.911,Z 409.908,A -85,B 0,C 180,E1 -3884.346,E2 -3884.346} C_VEL
LIN {X 0,Y 539.302,Z 398.096,A -85,B 0,C 180,E1 -3885.346,E2 -3885.346} C_VEL
LIN {X 0,Y 539.692,Z 385.139,A -85,B 0,C 180,E1 -3886.259,E2 -3886.259} C_VEL
LIN {X 0,Y 540.109,Z 371.818,A -85,B 0,C 180,E1 -3887.024,E2 -3887.024} C_VEL
LIN {X 0,Y 540.469,Z 358.26,A -85,B 0,C 180,E1 -3887.647,E2 -3887.647} C_VEL
LIN {X 0,Y 540.771,Z 343.308,A -85,B 0,C 180,E1 -3888.174,E2 -3888.174} C_VEL
LIN {X 0,Y 540.988,Z 328.853,A -85,B 0,C 180,E1 -3888.535,E2 -3888.535} C_VEL
LIN {X 0,Y 541.128,Z 306.107,A -85,B 0,C 180,E1 -3888.882,E2 -3888.882} C_VEL
LIN {X 0,Y 541.855,Z 172.302,A -85,B 0,C 180,E1 -3890.702,E2 -3890.702} C_VEL
LIN {X 0,Y 539.486,Z 160.958,A -85,B 0,C 180,E1 -3890.975,E2 -3890.975} C_VEL
LIN {X 0,Y 540.008,Z 142.188,A -85,B 0,C 180,E1 -3893.591,E2 -3893.591} C_VEL
LIN {X 0,Y 539.721,Z 136.674,A -85,B 0,C 180,E1 -3894.399,E2 -3894.399} C_VEL
LIN {X 0,Y 538.007,Z 129.343,A -85,B 0,C 180,E1 -3895.578,E2 -3895.578} C_VEL
LIN {X 0,Y 537.97,Z 129.098,A -85,B 0,C 180,E1 -3898.054,E2 -3898.054} C_VEL
LIN {X 0,Y 537.987,Z 129.083,A -85,B 0,C 180,E1 -3900.629,E2 -3900.629} C_VEL
LIN {X 0,Y 538.021,Z 129.092,A -85,B 0,C 180,E1 -3903.278,E2 -3903.278} C_VEL
LIN {X 0,Y 537.96,Z 129.094,A -85,B 0,C 180,E1 -3906.007,E2 -3906.007} C_VEL
LIN {X 0,Y 538.001,Z 129.097,A -85,B 0,C 180,E1 -3908.832,E2 -3908.832} C_VEL
LIN {X 0,Y 537.982,Z 129.093,A -85,B 0,C 180,E1 -3911.873,E2 -3911.873} C_VEL
LIN {X 0,Y 537.994,Z 129.094,A -85,B 0,C 180,E1 -3914.864,E2 -3914.864} C_VEL
LIN {X 0,Y 537.972,Z 129.095,A -85,B 0,C 180,E1 -3917.209,E2 -3917.209} C_VEL
LIN {X 0,Y 538.007,Z 129.083,A -85,B 0,C 180,E1 -3920.419,E2 -3920.419} C_VEL
LIN {X 0,Y 538.018,Z 129.091,A -85,B 0,C 180,E1 -3923.066,E2 -3923.066} C_VEL
LIN {X 0,Y 537.998,Z 129.088,A -85,B 0,C 180,E1 -3925.825,E2 -3925.825} C_VEL
LIN {X 0,Y 538.007,Z 129.083,A -85,B 0,C 180,E1 -3928.498,E2 -3928.498} C_VEL
LIN {X 0,Y 538.003,Z 129.089,A -85,B 0,C 180,E1 -3931.096,E2 -3931.096} C_VEL
LIN {X 0,Y 537.991,Z 129.091,A -85,B 0,C 180,E1 -3933.631,E2 -3933.631} C_VEL
LIN {X 0,Y 538.008,Z 129.093,A -85,B 0,C 180,E1 -3936.122,E2 -3936.122} C_VEL
LIN {X 0,Y 538.016,Z 129.089,A -85,B 0,C 180,E1 -3938.546,E2 -3938.546} C_VEL
LIN {X 0,Y 538.009,Z 129.087,A -85,B 0,C 180,E1 -3940.939,E2 -3940.939} C_VEL
LIN {X 0,Y 537.971,Z 129.094,A -85,B 0,C 180,E1 -3943.297,E2 -3943.297} C_VEL
LIN {X 0,Y 538.052,Z 129.084,A -85,B 0,C 180,E1 -3945.63,E2 -3945.63} C_VEL
LIN {X 0,Y 538.079,Z 129.08,A -85,B 0,C 180,E1 -3948.701,E2 -3948.701} C_VEL
LIN {X 0,Y 538.06,Z 129.085,A -85,B 0,C 180,E1 -3951.739,E2 -3951.739} C_VEL
LIN {X 0,Y 538.154,Z 129.07,A -85,B 0,C 180,E1 -3954.755,E2 -3954.755} C_VEL
LIN {X 0,Y 538.168,Z 129.072,A -85,B 0,C 180,E1 -3957.755,E2 -3957.755} C_VEL
LIN {X 0,Y 538.176,Z 129.068,A -85,B 0,C 180,E1 -3960.748,E2 -3960.748} C_VEL
LIN {X 0,Y 538.13,Z 129.073,A -85,B 0,C 180,E1 -3962.994,E2 -3962.994} C_VEL
LIN {X 0,Y 538.12,Z 129.076,A -85,B 0,C 180,E1 -3965.997,E2 -3965.997} C_VEL
LIN {X 0,Y 538.054,Z 129.086,A -85,B 0,C 180,E1 -3969.018,E2 -3969.018} C_VEL
LIN {X 0,Y 538.066,Z 129.082,A -85,B 0,C 180,E1 -3972.063,E2 -3972.063} C_VEL
LIN {X 0,Y 538.044,Z 129.088,A -85,B 0,C 180,E1 -3975.144,E2 -3975.144} C_VEL
LIN {X 0,Y 538.014,Z 129.089,A -85,B 0,C 180,E1 -3978.271,E2 -3978.271} C_VEL
LIN {X 0,Y 538.039,Z 129.088,A -85,B 0,C 180,E1 -3980.651,E2 -3980.651} C_VEL
LIN {X 0,Y 538.008,Z 129.089,A -85,B 0,C 180,E1 -3983.877,E2 -3983.877} C_VEL
LIN {X 0,Y 538.038,Z 129.085,A -85,B 0,C 180,E1 -3986.367,E2 -3986.367} C_VEL
LIN {X 0,Y 538.031,Z 129.091,A -85,B 0,C 180,E1 -3988.933,E2 -3988.933} C_VEL
LIN {X 0,Y 538.011,Z 129.081,A -85,B 0,C 180,E1 -3991.887,E2 -3991.887} C_VEL
LIN {X 0,Y 538.01,Z 129.089,A -85,B 0,C 180,E1 -3994.617,E2 -3994.617} C_VEL
LIN {X 0,Y 538.005,Z 129.09,A -85,B 0,C 180,E1 -3997.17,E2 -3997.17} C_VEL
LIN {X 0,Y 538.023,Z 129.083,A -85,B 0,C 180,E1 -3999.797,E2 -3999.797} C_VEL
LIN {X 0,Y 538.02,Z 129.091,A -85,B 0,C 180,E1 -4002.786,E2 -4002.786} C_VEL
LIN {X 0,Y 538.008,Z 129.086,A -85,B 0,C 180,E1 -4005.138,E2 -4005.138} C_VEL
LIN {X 0,Y 538.031,Z 129.094,A -85,B 0,C 180,E1 -4008.227,E2 -4008.227} C_VEL
LIN {X 0,Y 538.017,Z 129.086,A -85,B 0,C 180,E1 -4011.17,E2 -4011.17} C_VEL
LIN {X 0,Y 537.995,Z 129.094,A -85,B 0,C 180,E1 -4014.089,E2 -4014.089} C_VEL
LIN {X 0,Y 538.031,Z 129.083,A -85,B 0,C 180,E1 -4016.727,E2 -4016.727} C_VEL
LIN {X 0,Y 538.027,Z 129.087,A -85,B 0,C 180,E1 -4019.556,E2 -4019.556} C_VEL
LIN {X 0,Y 538.041,Z 129.076,A -85,B 0,C 180,E1 -4021.95,E2 -4021.95} C_VEL
LIN {X 0,Y 538.096,Z 129.299,A -85,B 0,C 180,E1 -4023.453,E2 -4023.453} C_VEL
LIN {X 0,Y 540.282,Z 139.511,A -85,B 0,C 180,E1 -4024.991,E2 -4024.991} C_VEL
LIN {X 0,Y 539.689,Z 160.441,A -85,B 0,C 180,E1 -4027.812,E2 -4027.812} C_VEL
LIN {X 0,Y 539.491,Z 169.828,A -85,B 0,C 180,E1 -4029.05,E2 -4029.05} C_VEL
LIN {X 0,Y 540.39,Z 174.652,A -85,B 0,C 180,E1 -4029.185,E2 -4029.185} C_VEL
LIN {X 0,Y 541.838,Z 182.201,A -85,B 0,C 180,E1 -4029.348,E2 -4029.348} C_VEL
LIN {X 0,Y 540.996,Z 336.081,A -85,B 0,C 180,E1 -4031.459,E2 -4031.459} C_VEL
LIN {X 0,Y 540.782,Z 351.502,A -85,B 0,C 180,E1 -4031.826,E2 -4031.826} C_VEL
LIN {X 0,Y 540.474,Z 365.612,A -85,B 0,C 180,E1 -4032.305,E2 -4032.305} C_VEL
LIN {X 0,Y 540.06,Z 380.611,A -85,B 0,C 180,E1 -4032.974,E2 -4032.974} C_VEL
LIN {X 0,Y 539.658,Z 394.096,A -85,B 0,C 180,E1 -4033.74,E2 -4033.74} C_VEL
LIN {X 0,Y 539.312,Z 407.157,A -85,B 0,C 180,E1 -4034.649,E2 -4034.649} C_VEL
LIN {X 0,Y 538.885,Z 419.169,A -85,B 0,C 180,E1 -4035.653,E2 -4035.653} C_VEL
LIN {X 0,Y 538.568,Z 430.65,A -85,B 0,C 180,E1 -4036.799,E2 -4036.799} C_VEL
LIN {X 0,Y 538.283,Z 440.311,A -85,B 0,C 180,E1 -4037.942,E2 -4037.942} C_VEL
LIN {X 0,Y 538.068,Z 449.797,A -85,B 0,C 180,E1 -4039.273,E2 -4039.273} C_VEL
LIN {X 0,Y 537.824,Z 457.697,A -85,B 0,C 180,E1 -4040.599,E2 -4040.599} C_VEL
LIN {X 0,Y 537.699,Z 465.07,A -85,B 0,C 180,E1 -4042.112,E2 -4042.112} C_VEL
LIN {X 0,Y 537.627,Z 470.385,A -85,B 0,C 180,E1 -4043.459,E2 -4043.459} C_VEL
LIN {X 0,Y 537.574,Z 474.385,A -85,B 0,C 180,E1 -4044.749,E2 -4044.749} C_VEL
LIN {X 0,Y 537.562,Z 477.886,A -85,B 0,C 180,E1 -4046.252,E2 -4046.252} C_VEL
LIN {X 0,Y 537.488,Z 480.188,A -85,B 0,C 180,E1 -4047.752,E2 -4047.752} C_VEL
LIN {X 0,Y 537.438,Z 481.347,A -85,B 0,C 180,E1 -4049.251,E2 -4049.251} C_VEL
LIN {X 0,Y 537.438,Z 481.346,A -85,B 0,C 180,E1 -4050.749,E2 -4050.749} C_VEL
LIN {X 0,Y 537.488,Z 480.184,A -85,B 0,C 180,E1 -4052.248,E2 -4052.248} C_VEL
LIN {X 0,Y 537.562,Z 477.881,A -85,B 0,C 180,E1 -4053.748,E2 -4053.748} C_VEL
LIN {X 0,Y 537.574,Z 474.386,A -85,B 0,C 180,E1 -4055.251,E2 -4055.251} C_VEL
LIN {X 0,Y 537.664,Z 469.604,A -85,B 0,C 180,E1 -4056.756,E2 -4056.756} C_VEL
LIN {X 0,Y 537.733,Z 463.397,A -85,B 0,C 180,E1 -4058.266,E2 -4058.266} C_VEL
LIN {X 0,Y 537.857,Z 455.599,A -85,B 0,C 180,E1 -4059.78,E2 -4059.78} C_VEL
LIN {X 0,Y 538.101,Z 447.305,A -85,B 0,C 180,E1 -4061.107,E2 -4061.107} C_VEL
LIN {X 0,Y 538.356,Z 437.308,A -85,B 0,C 180,E1 -4062.439,E2 -4062.439} C_VEL
LIN {X 0,Y 538.656,Z 427.08,A -85,B 0,C 180,E1 -4063.583,E2 -4063.583} C_VEL
LIN {X 0,Y 539.018,Z 414.893,A -85,B 0,C 180,E1 -4064.729,E2 -4064.729} C_VEL
LIN {X 0,Y 539.487,Z 401.352,A -85,B 0,C 180,E1 -4065.778,E2 -4065.778} C_VEL
LIN {X 0,Y 539.889,Z 387.719,A -85,B 0,C 180,E1 -4066.642,E2 -4066.642} C_VEL
LIN {X 0,Y 540.224,Z 373.622,A -85,B 0,C 180,E1 -4067.362,E2 -4067.362} C_VEL
LIN {X 0,Y 540.606,Z 359.115,A -85,B 0,C 180,E1 -4067.935,E2 -4067.935} C_VEL
LIN {X 0,Y 540.864,Z 344.256,A -85,B 0,C 180,E1 -4068.367,E2 -4068.367} C_VEL
LIN {X 0,Y 541.071,Z 329.201,A -85,B 0,C 180,E1 -4068.651,E2 -4068.651} C_VEL
LIN {X 0,Y 541.764,Z 181.491,A -85,B 0,C 180,E1 -4070.665,E2 -4070.665} C_VEL
LIN {X 0,Y 539.507,Z 170.145,A -85,B 0,C 180,E1 -4070.928,E2 -4070.928} C_VEL
LIN {X 0,Y 539.98,Z 149.978,A -85,B 0,C 180,E1 -4073.592,E2 -4073.592} C_VEL
LIN {X 0,Y 540.266,Z 139.511,A -85,B 0,C 180,E1 -4075.01,E2 -4075.01} C_VEL
LIN {X 0,Y 538.07,Z 129.206,A -85,B 0,C 180,E1 -4076.574,E2 -4076.574} C_VEL
LIN {X 0,Y 538.031,Z 129.089,A -85,B 0,C 180,E1 -4078.934,E2 -4078.934} C_VEL
LIN {X 0,Y 538.011,Z 129.08,A -85,B 0,C 180,E1 -4081.887,E2 -4081.887} C_VEL
LIN {X 0,Y 538.012,Z 129.091,A -85,B 0,C 180,E1 -4084.618,E2 -4084.618} C_VEL
LIN {X 0,Y 538.005,Z 129.09,A -85,B 0,C 180,E1 -4087.17,E2 -4087.17} C_VEL
LIN {X 0,Y 538.027,Z 129.089,A -85,B 0,C 180,E1 -4089.797,E2 -4089.797} C_VEL
LIN {X 0,Y 538.019,Z 129.086,A -85,B 0,C 180,E1 -4092.786,E2 -4092.786} C_VEL
LIN {X 0,Y 538.03,Z 129.093,A -85,B 0,C 180,E1 -4095.926,E2 -4095.926} C_VEL
LIN {X 0,Y 538.049,Z 129.082,A -85,B 0,C 180,E1 -4099.253,E2 -4099.253} C_VEL
LIN {X 0,Y 537.993,Z 129.093,A -85,B 0,C 180,E1 -4102.122,E2 -4102.122} C_VEL
LIN {X 0,Y 537.998,Z 129.09,A -85,B 0,C 180,E1 -4104.916,E2 -4104.916} C_VEL
LIN {X 0,Y 538.017,Z 129.083,A -85,B 0,C 180,E1 -4107.617,E2 -4107.617} C_VEL
LIN {X 0,Y 538.016,Z 129.087,A -85,B 0,C 180,E1 -4110.239,E2 -4110.239} C_VEL
LIN {X 0,Y 538.056,Z 129.085,A -85,B 0,C 180,E1 -4112.796,E2 -4112.796} C_VEL
LIN {X 0,Y 538.044,Z 129.092,A -85,B 0,C 180,E1 -4115.292,E2 -4115.292} C_VEL
LIN {X 0,Y 538.023,Z 129.086,A -85,B 0,C 180,E1 -4118.546,E2 -4118.546} C_VEL
LIN {X 0,Y 538.02,Z 129.093,A -85,B 0,C 180,E1 -4120.94,E2 -4120.94} C_VEL
LIN {X 0,Y 538.004,Z 129.09,A -85,B 0,C 180,E1 -4123.298,E2 -4123.298} C_VEL
LIN {X 0,Y 538.058,Z 129.082,A -85,B 0,C 180,E1 -4125.631,E2 -4125.631} C_VEL
LIN {X 0,Y 538.079,Z 129.087,A -85,B 0,C 180,E1 -4128.702,E2 -4128.702} C_VEL
LIN {X 0,Y 538.063,Z 129.08,A -85,B 0,C 180,E1 -4131.739,E2 -4131.739} C_VEL
LIN {X 0,Y 538.158,Z 129.074,A -85,B 0,C 180,E1 -4134.755,E2 -4134.755} C_VEL
LIN {X 0,Y 538.168,Z 129.066,A -85,B 0,C 180,E1 -4137.755,E2 -4137.755} C_VEL
LIN {X 0,Y 538.181,Z 129.069,A -85,B 0,C 180,E1 -4140.748,E2 -4140.748} C_VEL
LIN {X 0,Y 538.124,Z 129.073,A -85,B 0,C 180,E1 -4142.995,E2 -4142.995} C_VEL
LIN {X 0,Y 538.116,Z 129.079,A -85,B 0,C 180,E1 -4145.997,E2 -4145.997} C_VEL
LIN {X 0,Y 538.058,Z 129.08,A -85,B 0,C 180,E1 -4149.018,E2 -4149.018} C_VEL
LIN {X 0,Y 538.065,Z 129.089,A -85,B 0,C 180,E1 -4152.063,E2 -4152.063} C_VEL
LIN {X 0,Y 538.04,Z 129.081,A -85,B 0,C 180,E1 -4155.144,E2 -4155.144} C_VEL
LIN {X 0,Y 538.007,Z 129.092,A -85,B 0,C 180,E1 -4158.271,E2 -4158.271} C_VEL
LIN {X 0,Y 538.037,Z 129.083,A -85,B 0,C 180,E1 -4160.652,E2 -4160.652} C_VEL
LIN {X 0,Y 538.008,Z 129.094,A -85,B 0,C 180,E1 -4163.878,E2 -4163.878} C_VEL
LIN {X 0,Y 537.992,Z 129.092,A -85,B 0,C 180,E1 -4166.369,E2 -4166.369} C_VEL
LIN {X 0,Y 537.993,Z 129.091,A -85,B 0,C 180,E1 -4168.926,E2 -4168.926} C_VEL
LIN {X 0,Y 538.009,Z 129.08,A -85,B 0,C 180,E1 -4171.887,E2 -4171.887} C_VEL
LIN {X 0,Y 537.997,Z 129.087,A -85,B 0,C 180,E1 -4174.615,E2 -4174.615} C_VEL
LIN {X 0,Y 537.999,Z 129.095,A -85,B 0,C 180,E1 -4177.169,E2 -4177.169} C_VEL
LIN {X 0,Y 538.008,Z 129.081,A -85,B 0,C 180,E1 -4179.798,E2 -4179.798} C_VEL
LIN {X 0,Y 537.989,Z 129.081,A -85,B 0,C 180,E1 -4180.248,E2 -4180.248} C_VEL
LIN {X 0,Y 537.325,Z 129.166,A -85,B 0,C 180,E1 -4180.873,E2 -4180.873} C_VEL
LIN {X 0,Y 534.469,Z 129.533,A -85,B 0,C 180,E1 -4181.887,E2 -4181.887} C_VEL
LIN {X 0,Y 532.05,Z 129.84,A -85,B 0,C 180,E1 -4182.704,E2 -4182.704} C_VEL
LIN {X 0,Y 531.011,Z 129.969,A -85,B 0,C 180,E1 -4183.335,E2 -4183.335} C_VEL
LIN {X 0,Y 530.926,Z 129.976,A -85,B 0,C 180,E1 -4183.549,E2 -4183.549} C_VEL
LIN {X 0,Y 530.927,Z 129.967,A -85,B 0,C 180,E1 -4186.501,E2 -4186.501} C_VEL
LIN {X 0,Y 530.951,Z 129.967,A -85,B 0,C 180,E1 -4189.564,E2 -4189.564} C_VEL
LIN {X 0,Y 530.965,Z 129.97,A -85,B 0,C 180,E1 -4192.578,E2 -4192.578} C_VEL
LIN {X 0,Y 530.967,Z 129.97,A -85,B 0,C 180,E1 -4195.308,E2 -4195.308} C_VEL
LIN {X 0,Y 530.956,Z 129.97,A -85,B 0,C 180,E1 -4198.031,E2 -4198.031} C_VEL
LIN {X 0,Y 530.92,Z 129.972,A -85,B 0,C 180,E1 -4200.888,E2 -4200.888} C_VEL
LIN {X 0,Y 530.944,Z 129.962,A -85,B 0,C 180,E1 -4203.253,E2 -4203.253} C_VEL
LIN {X 0,Y 530.963,Z 130.155,A -85,B 0,C 180,E1 -4204.252,E2 -4204.252} C_VEL
LIN {X 0,Y 533.17,Z 140.208,A -85,B 0,C 180,E1 -4205.881,E2 -4205.881} C_VEL
LIN {X 0,Y 532.682,Z 157.206,A -85,B 0,C 180,E1 -4208.32,E2 -4208.32} C_VEL
LIN {X 0,Y 532.635,Z 161.003,A -85,B 0,C 180,E1 -4208.831,E2 -4208.831} C_VEL
LIN {X 0,Y 535.201,Z 174.054,A -85,B 0,C 180,E1 -4209.143,E2 -4209.143} C_VEL
LIN {X 0,Y 534.285,Z 326.781,A -85,B 0,C 180,E1 -4211.267,E2 -4211.267} C_VEL
LIN {X 0,Y 534.047,Z 342.134,A -85,B 0,C 180,E1 -4211.638,E2 -4211.638} C_VEL
LIN {X 0,Y 533.71,Z 357.402,A -85,B 0,C 180,E1 -4212.172,E2 -4212.172} C_VEL
LIN {X 0,Y 533.348,Z 370.115,A -85,B 0,C 180,E1 -4212.753,E2 -4212.753} C_VEL
LIN {X 0,Y 532.877,Z 383.756,A -85,B 0,C 180,E1 -4213.527,E2 -4213.527} C_VEL
LIN {X 0,Y 532.461,Z 396.667,A -85,B 0,C 180,E1 -4214.428,E2 -4214.428} C_VEL
LIN {X 0,Y 532.009,Z 408.993,A -85,B 0,C 180,E1 -4215.464,E2 -4215.464} C_VEL
LIN {X 0,Y 531.65,Z 420.505,A -85,B 0,C 180,E1 -4216.624,E2 -4216.624} C_VEL
LIN {X 0,Y 531.295,Z 430.195,A -85,B 0,C 180,E1 -4217.781,E2 -4217.781} C_VEL
LIN {X 0,Y 531.051,Z 439.694,A -85,B 0,C 180,E1 -4219.13,E2 -4219.13} C_VEL
LIN {X 0,Y 530.788,Z 448.609,A -85,B 0,C 180,E1 -4220.665,E2 -4220.665} C_VEL
LIN {X 0,Y 530.642,Z 454.991,A -85,B 0,C 180,E1 -4222.006,E2 -4222.006} C_VEL
LIN {X 0,Y 530.544,Z 460.642,A -85,B 0,C 180,E1 -4223.469,E2 -4223.469} C_VEL
LIN {X 0,Y 530.508,Z 464.329,A -85,B 0,C 180,E1 -4224.679,E2 -4224.679} C_VEL
LIN {X 0,Y 530.481,Z 467.853,A -85,B 0,C 180,E1 -4226.202,E2 -4226.202} C_VEL
LIN {X 0,Y 530.409,Z 470.188,A -85,B 0,C 180,E1 -4227.722,E2 -4227.722} C_VEL
LIN {X 0,Y 530.34,Z 471.385,A -85,B 0,C 180,E1 -4229.241,E2 -4229.241} C_VEL
LIN {X 0,Y 530.341,Z 471.405,A -85,B 0,C 180,E1 -4230.759,E2 -4230.759} C_VEL
LIN {X 0,Y 530.41,Z 470.287,A -85,B 0,C 180,E1 -4232.278,E2 -4232.278} C_VEL
LIN {X 0,Y 530.481,Z 468.029,A -85,B 0,C 180,E1 -4233.798,E2 -4233.798} C_VEL
LIN {X 0,Y 530.506,Z 464.578,A -85,B 0,C 180,E1 -4235.321,E2 -4235.321} C_VEL
LIN {X 0,Y 530.55,Z 459.854,A -85,B 0,C 180,E1 -4236.847,E2 -4236.847} C_VEL
LIN {X 0,Y 530.667,Z 453.732,A -85,B 0,C 180,E1 -4238.377,E2 -4238.377} C_VEL
LIN {X 0,Y 530.827,Z 446.025,A -85,B 0,C 180,E1 -4239.911,E2 -4239.911} C_VEL
LIN {X 0,Y 531.061,Z 437.807,A -85,B 0,C 180,E1 -4241.256,E2 -4241.256} C_VEL
LIN {X 0,Y 531.368,Z 427.913,A -85,B 0,C 180,E1 -4242.605,E2 -4242.605} C_VEL
LIN {X 0,Y 531.704,Z 417.769,A -85,B 0,C 180,E1 -4243.764,E2 -4243.764} C_VEL
LIN {X 0,Y 532.121,Z 405.698,A -85,B 0,C 180,E1 -4244.925,E2 -4244.925} C_VEL
LIN {X 0,Y 532.584,Z 393.579,A -85,B 0,C 180,E1 -4245.893,E2 -4245.893} C_VEL
LIN {X 0,Y 533.025,Z 380.463,A -85,B 0,C 180,E1 -4246.764,E2 -4246.764} C_VEL
LIN {X 0,Y 533.367,Z 367.958,A -85,B 0,C 180,E1 -4247.444,E2 -4247.444} C_VEL
LIN {X 0,Y 533.824,Z 353.335,A -85,B 0,C 180,E1 -4248.072,E2 -4248.072} C_VEL
LIN {X 0,Y 534.111,Z 337.735,A -85,B 0,C 180,E1 -4248.57,E2 -4248.57} C_VEL
LIN {X 0,Y 534.331,Z 323.383,A -85,B 0,C 180,E1 -4248.879,E2 -4248.879} C_VEL
LIN {X 0,Y 535.232,Z 173.946,A -85,B 0,C 180,E1 -4250.948,E2 -4250.948} C_VEL
LIN {X 0,Y 532.617,Z 161.059,A -85,B 0,C 180,E1 -4251.255,E2 -4251.255} C_VEL
LIN {X 0,Y 533.155,Z 143.659,A -85,B 0,C 180,E1 -4253.706,E2 -4253.706} C_VEL
LIN {X 0,Y 533.061,Z 139.401,A -85,B 0,C 180,E1 -4254.332,E2 -4254.332} C_VEL
LIN {X 0,Y 530.956,Z 130.178,A -85,B 0,C 180,E1 -4255.831,E2 -4255.831} C_VEL
LIN {X 0,Y 530.93,Z 129.975,A -85,B 0,C 180,E1 -4258.46,E2 -4258.46} C_VEL
LIN {X 0,Y 530.935,Z 129.966,A -85,B 0,C 180,E1 -4261.081,E2 -4261.081} C_VEL
LIN {X 0,Y 530.949,Z 129.97,A -85,B 0,C 180,E1 -4263.776,E2 -4263.776} C_VEL
LIN {X 0,Y 530.917,Z 129.973,A -85,B 0,C 180,E1 -4266.562,E2 -4266.562} C_VEL
LIN {X 0,Y 530.954,Z 129.966,A -85,B 0,C 180,E1 -4269.446,E2 -4269.446} C_VEL
LIN {X 0,Y 530.916,Z 129.976,A -85,B 0,C 180,E1 -4272.463,E2 -4272.463} C_VEL
LIN {X 0,Y 530.964,Z 129.967,A -85,B 0,C 180,E1 -4275.451,E2 -4275.451} C_VEL
LIN {X 0,Y 530.951,Z 129.971,A -85,B 0,C 180,E1 -4278.56,E2 -4278.56} C_VEL
LIN {X 0,Y 530.95,Z 129.965,A -85,B 0,C 180,E1 -4281.529,E2 -4281.529} C_VEL
LIN {X 0,Y 530.947,Z 129.975,A -85,B 0,C 180,E1 -4284.379,E2 -4284.379} C_VEL
LIN {X 0,Y 530.967,Z 129.954,A -85,B 0,C 180,E1 -4287.133,E2 -4287.133} C_VEL
LIN {X 0,Y 530.95,Z 129.962,A -85,B 0,C 180,E1 -4289.802,E2 -4289.802} C_VEL
LIN {X 0,Y 530.964,Z 129.973,A -85,B 0,C 180,E1 -4292.478,E2 -4292.478} C_VEL
LIN {X 0,Y 530.951,Z 129.965,A -85,B 0,C 180,E1 -4294.94,E2 -4294.94} C_VEL
LIN {X 0,Y 530.978,Z 129.969,A -85,B 0,C 180,E1 -4297.899,E2 -4297.899} C_VEL
LIN {X 0,Y 530.971,Z 129.965,A -85,B 0,C 180,E1 -4300.676,E2 -4300.676} C_VEL
LIN {X 0,Y 530.939,Z 129.969,A -85,B 0,C 180,E1 -4303.069,E2 -4303.069} C_VEL
LIN {X 0,Y 531.01,Z 129.959,A -85,B 0,C 180,E1 -4305.436,E2 -4305.436} C_VEL
LIN {X 0,Y 531.037,Z 129.958,A -85,B 0,C 180,E1 -4308.55,E2 -4308.55} C_VEL
LIN {X 0,Y 531.035,Z 129.959,A -85,B 0,C 180,E1 -4311.629,E2 -4311.629} C_VEL
LIN {X 0,Y 531.114,Z 129.947,A -85,B 0,C 180,E1 -4314.685,E2 -4314.685} C_VEL
LIN {X 0,Y 531.139,Z 129.946,A -85,B 0,C 180,E1 -4317.725,E2 -4317.725} C_VEL
LIN {X 0,Y 531.148,Z 129.943,A -85,B 0,C 180,E1 -4320.758,E2 -4320.758} C_VEL
LIN {X 0,Y 531.098,Z 129.95,A -85,B 0,C 180,E1 -4323.034,E2 -4323.034} C_VEL
LIN {X 0,Y 531.075,Z 129.953,A -85,B 0,C 180,E1 -4326.077,E2 -4326.077} C_VEL
LIN {X 0,Y 531.017,Z 129.963,A -85,B 0,C 180,E1 -4329.138,E2 -4329.138} C_VEL
LIN {X 0,Y 531.052,Z 129.958,A -85,B 0,C 180,E1 -4331.67,E2 -4331.67} C_VEL
LIN {X 0,Y 531.031,Z 129.962,A -85,B 0,C 180,E1 -4334.955,E2 -4334.955} C_VEL
LIN {X 0,Y 530.982,Z 129.965,A -85,B 0,C 180,E1 -4337.723,E2 -4337.723} C_VEL
LIN {X 0,Y 531.027,Z 129.957,A -85,B 0,C 180,E1 -4340.127,E2 -4340.127} C_VEL
LIN {X 0,Y 530.944,Z 129.971,A -85,B 0,C 180,E1 -4342.573,E2 -4342.573} C_VEL
LIN {X 0,Y 530.97,Z 129.967,A -85,B 0,C 180,E1 -4345.059,E2 -4345.059} C_VEL
LIN {X 0,Y 531.014,Z 129.96,A -85,B 0,C 180,E1 -4347.595,E2 -4347.595} C_VEL
LIN {X 0,Y 530.968,Z 129.967,A -85,B 0,C 180,E1 -4350.643,E2 -4350.643} C_VEL
LIN {X 0,Y 530.963,Z 129.955,A -85,B 0,C 180,E1 -4353.5,E2 -4353.5} C_VEL
LIN {X 0,Y 530.946,Z 129.971,A -85,B 0,C 180,E1 -4356.153,E2 -4356.153} C_VEL
LIN {X 0,Y 530.967,Z 129.966,A -85,B 0,C 180,E1 -4358.653,E2 -4358.653} C_VEL
LIN {X 0,Y 530.994,Z 129.958,A -85,B 0,C 180,E1 -4361.435,E2 -4361.435} C_VEL
LIN {X 0,Y 530.978,Z 129.966,A -85,B 0,C 180,E1 -4364.548,E2 -4364.548} C_VEL
LIN {X 0,Y 530.983,Z 129.967,A -85,B 0,C 180,E1 -4367.834,E2 -4367.834} C_VEL
LIN {X 0,Y 530.99,Z 129.964,A -85,B 0,C 180,E1 -4370.557,E2 -4370.557} C_VEL
LIN {X 0,Y 530.956,Z 129.97,A -85,B 0,C 180,E1 -4373.441,E2 -4373.441} C_VEL
LIN {X 0,Y 531,Z 129.96,A -85,B 0,C 180,E1 -4376.494,E2 -4376.494} C_VEL
LIN {X 0,Y 530.975,Z 129.963,A -85,B 0,C 180,E1 -4379.355,E2 -4379.355} C_VEL
LIN {X 0,Y 531.013,Z 129.951,A -85,B 0,C 180,E1 -4382.467,E2 -4382.467} C_VEL
LIN {X 0,Y 531.057,Z 130.173,A -85,B 0,C 180,E1 -4383.206,E2 -4383.206} C_VEL
LIN {X 0,Y 533.42,Z 140.947,A -85,B 0,C 180,E1 -4384.855,E2 -4384.855} C_VEL
LIN {X 0,Y 532.871,Z 160.376,A -85,B 0,C 180,E1 -4387.513,E2 -4387.513} C_VEL
LIN {X 0,Y 532.634,Z 170.011,A -85,B 0,C 180,E1 -4388.785,E2 -4388.785} C_VEL
LIN {X 0,Y 535.206,Z 183.517,A -85,B 0,C 180,E1 -4389.1,E2 -4389.1} C_VEL
LIN {X 0,Y 534.293,Z 335.803,A -85,B 0,C 180,E1 -4391.214,E2 -4391.214} C_VEL
LIN {X 0,Y 534.02,Z 351.436,A -85,B 0,C 180,E1 -4391.588,E2 -4391.588} C_VEL
LIN {X 0,Y 533.67,Z 366.78,A -85,B 0,C 180,E1 -4392.121,E2 -4392.121} C_VEL
LIN {X 0,Y 533.237,Z 380.544,A -85,B 0,C 180,E1 -4392.75,E2 -4392.75} C_VEL
LIN {X 0,Y 532.816,Z 394.03,A -85,B 0,C 180,E1 -4393.525,E2 -4393.525} C_VEL
LIN {X 0,Y 532.43,Z 406.533,A -85,B 0,C 180,E1 -4394.404,E2 -4394.404} C_VEL
LIN {X 0,Y 531.957,Z 419.102,A -85,B 0,C 180,E1 -4395.462,E2 -4395.462} C_VEL
LIN {X 0,Y 531.577,Z 430.583,A -85,B 0,C 180,E1 -4396.622,E2 -4396.622} C_VEL
LIN {X 0,Y 531.254,Z 440.243,A -85,B 0,C 180,E1 -4397.78,E2 -4397.78} C_VEL
LIN {X 0,Y 531.051,Z 449.73,A -85,B 0,C 180,E1 -4399.13,E2 -4399.13} C_VEL
LIN {X 0,Y 530.764,Z 457.63,A -85,B 0,C 180,E1 -4400.473,E2 -4400.473} C_VEL
LIN {X 0,Y 530.639,Z 465.004,A -85,B 0,C 180,E1 -4402.006,E2 -4402.006} C_VEL
LIN {X 0,Y 530.545,Z 470.628,A -85,B 0,C 180,E1 -4403.466,E2 -4403.466} C_VEL
LIN {X 0,Y 530.509,Z 474.326,A -85,B 0,C 180,E1 -4404.679,E2 -4404.679} C_VEL
LIN {X 0,Y 530.481,Z 477.837,A -85,B 0,C 180,E1 -4406.202,E2 -4406.202} C_VEL
LIN {X 0,Y 530.409,Z 480.146,A -85,B 0,C 180,E1 -4407.722,E2 -4407.722} C_VEL
LIN {X 0,Y 530.34,Z 481.308,A -85,B 0,C 180,E1 -4409.241,E2 -4409.241} C_VEL
LIN {X 0,Y 530.34,Z 481.307,A -85,B 0,C 180,E1 -4410.759,E2 -4410.759} C_VEL
LIN {X 0,Y 530.409,Z 480.142,A -85,B 0,C 180,E1 -4412.278,E2 -4412.278} C_VEL
LIN {X 0,Y 530.481,Z 477.832,A -85,B 0,C 180,E1 -4413.798,E2 -4413.798} C_VEL
LIN {X 0,Y 530.509,Z 474.327,A -85,B 0,C 180,E1 -4415.321,E2 -4415.321} C_VEL
LIN {X 0,Y 530.569,Z 469.537,A -85,B 0,C 180,E1 -4416.847,E2 -4416.847} C_VEL
LIN {X 0,Y 530.665,Z 463.33,A -85,B 0,C 180,E1 -4418.377,E2 -4418.377} C_VEL
LIN {X 0,Y 530.806,Z 455.532,A -85,B 0,C 180,E1 -4419.911,E2 -4419.911} C_VEL
LIN {X 0,Y 531.056,Z 447.238,A -85,B 0,C 180,E1 -4421.256,E2 -4421.256} C_VEL
LIN {X 0,Y 531.363,Z 437.241,A -85,B 0,C 180,E1 -4422.605,E2 -4422.605} C_VEL
LIN {X 0,Y 531.689,Z 427.013,A -85,B 0,C 180,E1 -4423.764,E2 -4423.764} C_VEL
LIN {X 0,Y 532.109,Z 414.827,A -85,B 0,C 180,E1 -4424.925,E2 -4424.925} C_VEL
LIN {X 0,Y 532.582,Z 402.595,A -85,B 0,C 180,E1 -4425.891,E2 -4425.891} C_VEL
LIN {X 0,Y 532.992,Z 389.275,A -85,B 0,C 180,E1 -4426.765,E2 -4426.765} C_VEL
LIN {X 0,Y 533.404,Z 374.576,A -85,B 0,C 180,E1 -4427.541,E2 -4427.541} C_VEL
LIN {X 0,Y 533.815,Z 360.358,A -85,B 0,C 180,E1 -4428.122,E2 -4428.122} C_VEL
LIN {X 0,Y 534.085,Z 346.11,A -85,B 0,C 180,E1 -4428.556,E2 -4428.556} C_VEL
LIN {X 0,Y 534.321,Z 331.364,A -85,B 0,C 180,E1 -4428.859,E2 -4428.859} C_VEL
LIN {X 0,Y 535.18,Z 182.768,A -85,B 0,C 180,E1 -4430.912,E2 -4430.912} C_VEL
LIN {X 0,Y 532.63,Z 169.891,A -85,B 0,C 180,E1 -4431.223,E2 -4431.223} C_VEL
LIN {X 0,Y 533.164,Z 149.917,A -85,B 0,C 180,E1 -4433.912,E2 -4433.912} C_VEL
LIN {X 0,Y 533.401,Z 140.948,A -85,B 0,C 180,E1 -4435.146,E2 -4435.146} C_VEL
LIN {X 0,Y 531.046,Z 130.056,A -85,B 0,C 180,E1 -4436.834,E2 -4436.834} C_VEL
LIN {X 0,Y 530.982,Z 129.966,A -85,B 0,C 180,E1 -4439.323,E2 -4439.323} C_VEL
LIN {X 0,Y 530.966,Z 129.957,A -85,B 0,C 180,E1 -4442.1,E2 -4442.1} C_VEL
LIN {X 0,Y 530.97,Z 129.967,A -85,B 0,C 180,E1 -4444.851,E2 -4444.851} C_VEL
LIN {X 0,Y 530.966,Z 129.969,A -85,B 0,C 180,E1 -4447.508,E2 -4447.508} C_VEL
LIN {X 0,Y 530.983,Z 129.966,A -85,B 0,C 180,E1 -4450.433,E2 -4450.433} C_VEL
LIN {X 0,Y 530.961,Z 129.967,A -85,B 0,C 180,E1 -4453.281,E2 -4453.281} C_VEL
LIN {X 0,Y 530.982,Z 129.968,A -85,B 0,C 180,E1 -4455.622,E2 -4455.622} C_VEL
LIN {X 0,Y 530.994,Z 129.957,A -85,B 0,C 180,E1 -4458.565,E2 -4458.565} C_VEL
LIN {X 0,Y 530.958,Z 129.971,A -85,B 0,C 180,E1 -4461.529,E2 -4461.529} C_VEL
LIN {X 0,Y 530.955,Z 129.965,A -85,B 0,C 180,E1 -4464.38,E2 -4464.38} C_VEL
LIN {X 0,Y 530.967,Z 129.956,A -85,B 0,C 180,E1 -4467.133,E2 -4467.133} C_VEL
LIN {X 0,Y 530.962,Z 129.968,A -85,B 0,C 180,E1 -4469.803,E2 -4469.803} C_VEL
LIN {X 0,Y 531.013,Z 129.96,A -85,B 0,C 180,E1 -4472.468,E2 -4472.468} C_VEL
LIN {X 0,Y 531.001,Z 129.963,A -85,B 0,C 180,E1 -4474.942,E2 -4474.942} C_VEL
LIN {X 0,Y 530.973,Z 129.963,A -85,B 0,C 180,E1 -4478.247,E2 -4478.247} C_VEL
LIN {X 0,Y 530.984,Z 129.966,A -85,B 0,C 180,E1 -4480.677,E2 -4480.677} C_VEL
LIN {X 0,Y 530.965,Z 129.97,A -85,B 0,C 180,E1 -4483.07,E2 -4483.07} C_VEL
LIN {X 0,Y 531.016,Z 129.961,A -85,B 0,C 180,E1 -4485.436,E2 -4485.436} C_VEL
LIN {X 0,Y 531.037,Z 129.962,A -85,B 0,C 180,E1 -4488.55,E2 -4488.55} C_VEL
LIN {X 0,Y 531.038,Z 129.955,A -85,B 0,C 180,E1 -4491.629,E2 -4491.629} C_VEL
LIN {X 0,Y 531.118,Z 129.952,A -85,B 0,C 180,E1 -4494.685,E2 -4494.685} C_VEL
LIN {X 0,Y 531.14,Z 129.941,A -85,B 0,C 180,E1 -4497.725,E2 -4497.725} C_VEL
LIN {X 0,Y 531.151,Z 129.944,A -85,B 0,C 180,E1 -4500.758,E2 -4500.758} C_VEL
LIN {X 0,Y 531.091,Z 129.948,A -85,B 0,C 180,E1 -4503.034,E2 -4503.034} C_VEL
LIN {X 0,Y 531.071,Z 129.958,A -85,B 0,C 180,E1 -4506.077,E2 -4506.077} C_VEL
LIN {X 0,Y 531.018,Z 129.956,A -85,B 0,C 180,E1 -4509.138,E2 -4509.138} C_VEL
LIN {X 0,Y 531.052,Z 129.958,A -85,B 0,C 180,E1 -4511.671,E2 -4511.671} C_VEL
LIN {X 0,Y 531.025,Z 129.955,A -85,B 0,C 180,E1 -4514.952,E2 -4514.952} C_VEL
LIN {X 0,Y 530.97,Z 129.965,A -85,B 0,C 180,E1 -4518.522,E2 -4518.522} C_VEL
LIN {X 0,Y 530.999,Z 129.959,A -85,B 0,C 180,E1 -4520.938,E2 -4520.938} C_VEL
LIN {X 0,Y 530.952,Z 129.968,A -85,B 0,C 180,E1 -4524.226,E2 -4524.226} C_VEL
LIN {X 0,Y 530.958,Z 129.966,A -85,B 0,C 180,E1 -4526.746,E2 -4526.746} C_VEL
LIN {X 0,Y 530.962,Z 129.97,A -85,B 0,C 180,E1 -4529.324,E2 -4529.324} C_VEL
LIN {X 0,Y 530.963,Z 129.955,A -85,B 0,C 180,E1 -4532.1,E2 -4532.1} C_VEL
LIN {X 0,Y 530.958,Z 129.965,A -85,B 0,C 180,E1 -4534.849,E2 -4534.849} C_VEL
LIN {X 0,Y 530.963,Z 129.971,A -85,B 0,C 180,E1 -4537.508,E2 -4537.508} C_VEL
LIN {X 0,Y 530.951,Z 129.957,A -85,B 0,C 180,E1 -4540.436,E2 -4540.436} C_VEL
LIN {X 0,Y 530.926,Z 129.976,A -85,B 0,C 180,E1 -4543.549,E2 -4543.549} C_VEL
LIN {X 0,Y 530.262,Z 130.054,A -85,B 0,C 180,E1 -4544.182,E2 -4544.182} C_VEL
LIN {X 0,Y 527.42,Z 130.41,A -85,B 0,C 180,E1 -4545.211,E2 -4545.211} C_VEL
LIN {X 0,Y 525.012,Z 130.707,A -85,B 0,C 180,E1 -4546.04,E2 -4546.04} C_VEL
LIN {X 0,Y 523.968,Z 130.836,A -85,B 0,C 180,E1 -4546.68,E2 -4546.68} C_VEL
LIN {X 0,Y 523.878,Z 130.847,A -85,B 0,C 180,E1 -4546.896,E2 -4546.896} C_VEL
LIN {X 0,Y 523.913,Z 130.84,A -85,B 0,C 180,E1 -4549.917,E2 -4549.917} C_VEL
LIN {X 0,Y 523.902,Z 130.853,A -85,B 0,C 180,E1 -4552.867,E2 -4552.867} C_VEL
LIN {X 0,Y 523.911,Z 130.846,A -85,B 0,C 180,E1 -4555.708,E2 -4555.708} C_VEL
LIN {X 0,Y 523.907,Z 130.851,A -85,B 0,C 180,E1 -4558.455,E2 -4558.455} C_VEL
LIN {X 0,Y 523.872,Z 130.855,A -85,B 0,C 180,E1 -4561.121,E2 -4561.121} C_VEL
LIN {X 0,Y 523.926,Z 131.008,A -85,B 0,C 180,E1 -4563.994,E2 -4563.994} C_VEL
LIN {X 0,Y 526.291,Z 141.688,A -85,B 0,C 180,E1 -4565.756,E2 -4565.756} C_VEL
LIN {X 0,Y 525.852,Z 157.274,A -85,B 0,C 180,E1 -4568.024,E2 -4568.024} C_VEL
LIN {X 0,Y 525.783,Z 161.196,A -85,B 0,C 180,E1 -4568.549,E2 -4568.549} C_VEL
LIN {X 0,Y 528.597,Z 175.123,A -85,B 0,C 180,E1 -4568.883,E2 -4568.883} C_VEL
LIN {X 0,Y 527.59,Z 326.528,A -85,B 0,C 180,E1 -4571.013,E2 -4571.013} C_VEL
LIN {X 0,Y 527.3,Z 342.221,A -85,B 0,C 180,E1 -4571.395,E2 -4571.395} C_VEL
LIN {X 0,Y 526.965,Z 357.482,A -85,B 0,C 180,E1 -4571.936,E2 -4571.936} C_VEL
LIN {X 0,Y 526.544,Z 370.195,A -85,B 0,C 180,E1 -4572.523,E2 -4572.523} C_VEL
LIN {X 0,Y 526.052,Z 383.832,A -85,B 0,C 180,E1 -4573.307,E2 -4573.307} C_VEL
LIN {X 0,Y 525.597,Z 396.706,A -85,B 0,C 180,E1 -4574.216,E2 -4574.216} C_VEL
LIN {X 0,Y 525.094,Z 409.066,A -85,B 0,C 180,E1 -4575.268,E2 -4575.268} C_VEL
LIN {X 0,Y 524.679,Z 420.578,A -85,B 0,C 180,E1 -4576.443,E2 -4576.443} C_VEL
LIN {X 0,Y 524.312,Z 430.267,A -85,B 0,C 180,E1 -4577.616,E2 -4577.616} C_VEL
LIN {X 0,Y 524.035,Z 439.764,A -85,B 0,C 180,E1 -4578.982,E2 -4578.982} C_VEL
LIN {X 0,Y 523.765,Z 447.674,A -85,B 0,C 180,E1 -4580.344,E2 -4580.344} C_VEL
LIN {X 0,Y 523.566,Z 455.061,A -85,B 0,C 180,E1 -4581.897,E2 -4581.897} C_VEL
LIN {X 0,Y 523.467,Z 461.002,A -85,B 0,C 180,E1 -4583.471,E2 -4583.471} C_VEL
LIN {X 0,Y 523.445,Z 464.397,A -85,B 0,C 180,E1 -4584.607,E2 -4584.607} C_VEL
LIN {X 0,Y 523.402,Z 467.921,A -85,B 0,C 180,E1 -4586.15,E2 -4586.15} C_VEL
LIN {X 0,Y 523.333,Z 470.255,A -85,B 0,C 180,E1 -4587.691,E2 -4587.691} C_VEL
LIN {X 0,Y 523.246,Z 471.452,A -85,B 0,C 180,E1 -4589.23,E2 -4589.23} C_VEL
LIN {X 0,Y 523.247,Z 471.471,A -85,B 0,C 180,E1 -4590.77,E2 -4590.77} C_VEL
LIN {X 0,Y 523.333,Z 470.352,A -85,B 0,C 180,E1 -4592.309,E2 -4592.309} C_VEL
LIN {X 0,Y 523.402,Z 468.094,A -85,B 0,C 180,E1 -4593.85,E2 -4593.85} C_VEL
LIN {X 0,Y 523.442,Z 464.643,A -85,B 0,C 180,E1 -4595.393,E2 -4595.393} C_VEL
LIN {X 0,Y 523.482,Z 459.918,A -85,B 0,C 180,E1 -4596.94,E2 -4596.94} C_VEL
LIN {X 0,Y 523.613,Z 453.795,A -85,B 0,C 180,E1 -4598.49,E2 -4598.49} C_VEL
LIN {X 0,Y 523.79,Z 446.088,A -85,B 0,C 180,E1 -4600.045,E2 -4600.045} C_VEL
LIN {X 0,Y 524.034,Z 437.87,A -85,B 0,C 180,E1 -4601.409,E2 -4601.409} C_VEL
LIN {X 0,Y 524.37,Z 427.975,A -85,B 0,C 180,E1 -4602.776,E2 -4602.776} C_VEL
LIN {X 0,Y 524.768,Z 417.831,A -85,B 0,C 180,E1 -4603.95,E2 -4603.95} C_VEL
LIN {X 0,Y 525.239,Z 405.758,A -85,B 0,C 180,E1 -4605.125,E2 -4605.125} C_VEL
LIN {X 0,Y 525.738,Z 392.499,A -85,B 0,C 180,E1 -4606.194,E2 -4606.194} C_VEL
LIN {X 0,Y 526.293,Z 378.939,A -85,B 0,C 180,E1 -4607.085,E2 -4607.085} C_VEL
LIN {X 0,Y 526.739,Z 364.004,A -85,B 0,C 180,E1 -4607.871,E2 -4607.871} C_VEL
LIN {X 0,Y 527.175,Z 348.732,A -85,B 0,C 180,E1 -4608.484,E2 -4608.484} C_VEL
LIN {X 0,Y 527.465,Z 334.126,A -85,B 0,C 180,E1 -4608.913,E2 -4608.913} C_VEL
LIN {X 0,Y 527.693,Z 318.177,A -85,B 0,C 180,E1 -4609.212,E2 -4609.212} C_VEL
LIN {X 0,Y 528.517,Z 173.821,A -85,B 0,C 180,E1 -4611.229,E2 -4611.229} C_VEL
LIN {X 0,Y 525.788,Z 161.212,A -85,B 0,C 180,E1 -4611.541,E2 -4611.541} C_VEL
LIN {X 0,Y 526.123,Z 150.946,A -85,B 0,C 180,E1 -4612.979,E2 -4612.979} C_VEL
LIN {X 0,Y 526.346,Z 142.297,A -85,B 0,C 180,E1 -4614.242,E2 -4614.242} C_VEL
LIN {X 0,Y 523.954,Z 131.33,A -85,B 0,C 180,E1 -4616.013,E2 -4616.013} C_VEL
LIN {X 0,Y 523.882,Z 130.844,A -85,B 0,C 180,E1 -4616.277,E2 -4616.277} C_VEL
LIN {X 0,Y 523.872,Z 130.857,A -85,B 0,C 180,E1 -4618.879,E2 -4618.879} C_VEL
LIN {X 0,Y 523.905,Z 130.85,A -85,B 0,C 180,E1 -4621.545,E2 -4621.545} C_VEL
LIN {X 0,Y 523.911,Z 130.845,A -85,B 0,C 180,E1 -4624.292,E2 -4624.292} C_VEL
LIN {X 0,Y 523.88,Z 130.851,A -85,B 0,C 180,E1 -4627.674,E2 -4627.674} C_VEL
LIN {X 0,Y 523.914,Z 130.84,A -85,B 0,C 180,E1 -4630.126,E2 -4630.126} C_VEL
LIN {X 0,Y 523.881,Z 130.848,A -85,B 0,C 180,E1 -4633.171,E2 -4633.171} C_VEL
LIN {X 0,Y 523.92,Z 130.844,A -85,B 0,C 180,E1 -4635.77,E2 -4635.77} C_VEL
LIN {X 0,Y 523.888,Z 130.843,A -85,B 0,C 180,E1 -4638.903,E2 -4638.903} C_VEL
LIN {X 0,Y 523.911,Z 130.842,A -85,B 0,C 180,E1 -4641.898,E2 -4641.898} C_VEL
LIN {X 0,Y 523.918,Z 130.845,A -85,B 0,C 180,E1 -4644.913,E2 -4644.913} C_VEL
LIN {X 0,Y 523.935,Z 130.828,A -85,B 0,C 180,E1 -4647.68,E2 -4647.68} C_VEL
LIN {X 0,Y 523.937,Z 130.846,A -85,B 0,C 180,E1 -4650.68,E2 -4650.68} C_VEL
LIN {X 0,Y 523.903,Z 130.847,A -85,B 0,C 180,E1 -4653.725,E2 -4653.725} C_VEL
LIN {X 0,Y 523.909,Z 130.851,A -85,B 0,C 180,E1 -4656.269,E2 -4656.269} C_VEL
LIN {X 0,Y 523.942,Z 130.84,A -85,B 0,C 180,E1 -4658.766,E2 -4658.766} C_VEL
LIN {X 0,Y 523.93,Z 130.84,A -85,B 0,C 180,E1 -4661.22,E2 -4661.22} C_VEL
LIN {X 0,Y 523.883,Z 130.852,A -85,B 0,C 180,E1 -4663.637,E2 -4663.637} C_VEL
LIN {X 0,Y 523.925,Z 130.846,A -85,B 0,C 180,E1 -4666.028,E2 -4666.028} C_VEL
LIN {X 0,Y 523.994,Z 130.835,A -85,B 0,C 180,E1 -4669.177,E2 -4669.177} C_VEL
LIN {X 0,Y 523.978,Z 130.836,A -85,B 0,C 180,E1 -4672.292,E2 -4672.292} C_VEL
LIN {X 0,Y 524.075,Z 130.824,A -85,B 0,C 180,E1 -4674.614,E2 -4674.614} C_VEL
LIN {X 0,Y 524.111,Z 130.821,A -85,B 0,C 180,E1 -4677.694,E2 -4677.694} C_VEL
LIN {X 0,Y 524.119,Z 130.819,A -85,B 0,C 180,E1 -4680.768,E2 -4680.768} C_VEL
LIN {X 0,Y 524.04,Z 130.829,A -85,B 0,C 180,E1 -4683.075,E2 -4683.075} C_VEL
LIN {X 0,Y 524.035,Z 130.829,A -85,B 0,C 180,E1 -4686.159,E2 -4686.159} C_VEL
LIN {X 0,Y 523.987,Z 130.837,A -85,B 0,C 180,E1 -4689.262,E2 -4689.262} C_VEL
LIN {X 0,Y 524.002,Z 130.836,A -85,B 0,C 180,E1 -4691.737,E2 -4691.737} C_VEL
LIN {X 0,Y 523.994,Z 130.837,A -85,B 0,C 180,E1 -4695.051,E2 -4695.051} C_VEL
LIN {X 0,Y 523.946,Z 130.841,A -85,B 0,C 180,E1 -4697.97,E2 -4697.97} C_VEL
LIN {X 0,Y 523.974,Z 130.837,A -85,B 0,C 180,E1 -4700.41,E2 -4700.41} C_VEL
LIN {X 0,Y 523.91,Z 130.852,A -85,B 0,C 180,E1 -4702.894,E2 -4702.894} C_VEL
LIN {X 0,Y 523.916,Z 130.842,A -85,B 0,C 180,E1 -4705.42,E2 -4705.42} C_VEL
LIN {X 0,Y 523.966,Z 130.838,A -85,B 0,C 180,E1 -4707.999,E2 -4707.999} C_VEL
LIN {X 0,Y 523.94,Z 130.838,A -85,B 0,C 180,E1 -4710.853,E2 -4710.853} C_VEL
LIN {X 0,Y 523.931,Z 130.83,A -85,B 0,C 180,E1 -4713.729,E2 -4713.729} C_VEL
LIN {X 0,Y 523.905,Z 130.851,A -85,B 0,C 180,E1 -4716.401,E2 -4716.401} C_VEL
LIN {X 0,Y 523.921,Z 130.839,A -85,B 0,C 180,E1 -4719.085,E2 -4719.085} C_VEL
LIN {X 0,Y 523.952,Z 130.84,A -85,B 0,C 180,E1 -4722.119,E2 -4722.119} C_VEL
LIN {X 0,Y 523.945,Z 130.837,A -85,B 0,C 180,E1 -4725.31,E2 -4725.31} C_VEL
LIN {X 0,Y 523.957,Z 130.841,A -85,B 0,C 180,E1 -4728.69,E2 -4728.69} C_VEL
LIN {X 0,Y 523.92,Z 130.842,A -85,B 0,C 180,E1 -4731.08,E2 -4731.08} C_VEL
LIN {X 0,Y 523.901,Z 130.85,A -85,B 0,C 180,E1 -4733.825,E2 -4733.825} C_VEL
LIN {X 0,Y 523.942,Z 130.838,A -85,B 0,C 180,E1 -4736.635,E2 -4736.635} C_VEL
LIN {X 0,Y 523.957,Z 130.837,A -85,B 0,C 180,E1 -4739.356,E2 -4739.356} C_VEL
LIN {X 0,Y 523.978,Z 130.825,A -85,B 0,C 180,E1 -4742.281,E2 -4742.281} C_VEL
LIN {X 0,Y 524.031,Z 131.089,A -85,B 0,C 180,E1 -4742.96,E2 -4742.96} C_VEL
LIN {X 0,Y 526.543,Z 142.383,A -85,B 0,C 180,E1 -4744.715,E2 -4744.715} C_VEL
LIN {X 0,Y 526.058,Z 160.311,A -85,B 0,C 180,E1 -4747.205,E2 -4747.205} C_VEL
LIN {X 0,Y 525.769,Z 170.093,A -85,B 0,C 180,E1 -4748.501,E2 -4748.501} C_VEL
LIN {X 0,Y 528.567,Z 183.943,A -85,B 0,C 180,E1 -4748.831,E2 -4748.831} C_VEL
LIN {X 0,Y 527.558,Z 336.3,A -85,B 0,C 180,E1 -4750.977,E2 -4750.977} C_VEL
LIN {X 0,Y 527.257,Z 351.369,A -85,B 0,C 180,E1 -4751.343,E2 -4751.343} C_VEL
LIN {X 0,Y 526.899,Z 366.713,A -85,B 0,C 180,E1 -4751.883,E2 -4751.883} C_VEL
LIN {X 0,Y 526.43,Z 380.477,A -85,B 0,C 180,E1 -4752.519,E2 -4752.519} C_VEL
LIN {X 0,Y 525.961,Z 393.963,A -85,B 0,C 180,E1 -4753.304,E2 -4753.304} C_VEL
LIN {X 0,Y 525.525,Z 407.187,A -85,B 0,C 180,E1 -4754.249,E2 -4754.249} C_VEL
LIN {X 0,Y 524.996,Z 420.106,A -85,B 0,C 180,E1 -4755.364,E2 -4755.364} C_VEL
LIN {X 0,Y 524.572,Z 432.282,A -85,B 0,C 180,E1 -4756.638,E2 -4756.638} C_VEL
LIN {X 0,Y 524.137,Z 443.105,A -85,B 0,C 180,E1 -4758.005,E2 -4758.005} C_VEL
LIN {X 0,Y 523.926,Z 452.113,A -85,B 0,C 180,E1 -4759.371,E2 -4759.371} C_VEL
LIN {X 0,Y 523.676,Z 459.583,A -85,B 0,C 180,E1 -4760.732,E2 -4760.732} C_VEL
LIN {X 0,Y 523.515,Z 466.552,A -85,B 0,C 180,E1 -4762.285,E2 -4762.285} C_VEL
LIN {X 0,Y 523.441,Z 472.029,A -85,B 0,C 180,E1 -4763.834,E2 -4763.834} C_VEL
LIN {X 0,Y 523.323,Z 476.169,A -85,B 0,C 180,E1 -4765.378,E2 -4765.378} C_VEL
LIN {X 0,Y 523.358,Z 479.071,A -85,B 0,C 180,E1 -4766.921,E2 -4766.921} C_VEL
LIN {X 0,Y 523.272,Z 480.801,A -85,B 0,C 180,E1 -4768.461,E2 -4768.461} C_VEL
LIN {X 0,Y 523.243,Z 481.395,A -85,B 0,C 180,E1 -4770,E2 -4770} C_VEL
LIN {X 0,Y 523.272,Z 480.799,A -85,B 0,C 180,E1 -4771.539,E2 -4771.539} C_VEL
LIN {X 0,Y 523.358,Z 479.066,A -85,B 0,C 180,E1 -4773.079,E2 -4773.079} C_VEL
LIN {X 0,Y 523.323,Z 476.167,A -85,B 0,C 180,E1 -4774.622,E2 -4774.622} C_VEL
LIN {X 0,Y 523.451,Z 472.034,A -85,B 0,C 180,E1 -4776.166,E2 -4776.166} C_VEL
LIN {X 0,Y 523.515,Z 466.553,A -85,B 0,C 180,E1 -4777.715,E2 -4777.715} C_VEL
LIN {X 0,Y 523.676,Z 459.577,A -85,B 0,C 180,E1 -4779.268,E2 -4779.268} C_VEL
